REGION Network 4: Block description — Section 3.6 to 4
   // ▂▂▂▂▂▂▂▂▂▂▂▂▂▂▂▂▂▂▂▂▂▂▂▂▂▂▂▂▂▂▂▂▂▂▂▂▂▂▂▂▂▂▂▂
   // 3.6     Operating modes
   // 
   // 
   // This module FC11011_StdDevValve3Way supports various operating modes:
   // 
   //    •   Automatic/manual mode
   // 
   //    •   Interlock bypass mode
   // 
   //    •   Simulation mode
   // 
   //    •   Remote/local mode
   // 
   //    •   Faceplate disabled mode
   // 
   // Examining these in turn:   
   // 
   // 
   // 
   // ▁▁▁▁▁▁▁▁▁▁▁▁▁▁▁▁▁▁▁▁▁▁▁▁▁▁▁▁▁▁▁▁▁▁▁▁▁▁▁▁▁▁▁▁
   // 3.6.1    Automatic and manual modes
   // 
   // 
   // Under normal operation, the valve is in automatic mode and is controlled directly by the 
   // Controller software (usually, sequential or continuous logic); however, it is possible for the 
   // operator to take direct control of the valve by switching it to manual mode.
   // 
   // If manual mode is active, the valve will be energised and deenergised directly at the command 
   // of the operator and will ignore any automatic mode energise and deenergise requests.
   // 
   // If the valve is operating under automatic mode, the manual energise/deenergise request follows 
   // that of the automatic mode; this ensures that the valve remains in the same state when initially 
   // switched from automatic mode to manual mode, referred to as bumpless transfer. This approach 
   // minimises any disturbance to the process should the valve be inadvertently switched to manual 
   // mode.
   // 
   // The following data points are associated with automatic/manual mode:
   // 
   //  DATA STRUCTURE    UT11011_St_DevValve3Way
   //  ――――――――――――――――――――――――――――――――――――――――――
   //  SIGNAL         FUNCTION               TYPE     DETAILS
   //  ――――――――――――――――――――――――――――――――――――――――――
   //  CONFIG_MAN_DIS     Prevents manual mode being       Bool  1 = no manual mode
   //            activated under all circumstances            0 = manual permitted
   //  ――――――――――――――――――――――――――――――――――――――――――
   // 
   //  DATA STRUCTURE    UT31011_Dy_DevValve3Way
   //  ――――――――――――――――――――――――――――――――――――――――――
   //  SIGNAL         FUNCTION               TYPE     DETAILS
   //  ――――――――――――――――――――――――――――――――――――――――――
   //  Mode_AutMan     Identifies the operating mode of     Bool  1 = automatic mode
   //            the valve.                   0 = manual mode
   // 
   //  ctrl_Aut_EngDeng    Causes the valve to energise and         Bool  1 = energise valve
   //            deenergise if auto mode is active          0 = deenergise valve
   // 
   //  ctrl_Man_EngDeng   Causes the valve to energise and         Bool  1 = energise valve
   //            deenergise if man mode is active          0 = deenergise valve
   // 
   //  status_Aut      The valve is in automatic mode      Bool  1 = auto mode
   //                                  0 = no in auto
   // 
   //  status_Man       The valve is in manual mode     Bool  1 = manual mode
   //                                  0 = no in manual
   //  ――――――――――――――――――――――――――――――――――――――――――
   // 
   // Manual mode can only be activated by the operator via a faceplate available at the supervisory 
   // system (SCADA/HMI). 
   // 
   // 
   // 
   // ▁▁▁▁▁▁▁▁▁▁▁▁▁▁▁▁▁▁▁▁▁▁▁▁▁▁▁▁▁▁▁▁▁▁▁▁▁▁▁▁▁▁▁▁
   // 3.6.2    Interlock bypass mode
   // 
   // 
   // All interlock signals (TRIP, INTERLOCK or PERMISSIVE) can be overridden (bypassed). The bypass 
   // signal is a single signal that, if active, overrides and deactivates any TRIP, INTERLOCK or 
   // PERMISSIVE signal that may have been activated.
   // 
   // It is possible to permanently disable the bypass mode for any given valve (preventing the 
   // operator from activating it).
   // 
   // The following data points are associated with the bypass mode:
   // 
   //  DATA STRUCTURE    UT11011_St_DevValve3Way
   //  ――――――――――――――――――――――――――――――――――――――――――
   //  SIGNAL       FUNCTION                TYPE     DETAILS
   //  ――――――――――――――――――――――――――――――――――――――――――
   //  CONFIG_BYPASS_DIS    Prevents bypass mode being      Bool     1 = no bypass mode
   //             activated under all circumstances         0 = bypass permitted
   //  ――――――――――――――――――――――――――――――――――――――――――
   // 
   //  DATA STRUCTURE    UT31011_Dy_DevValve3Way
   //  ――――――――――――――――――――――――――――――――――――――――――
   //  SIGNAL         FUNCTION                TYPE     DETAILS
   //  ――――――――――――――――――――――――――――――――――――――――――
   //  mode_BypassOn   Activates bypass mode, if active, any    Bool     1 = bypass mode on
   //            TRIP, INTERLOCK or PERMISSIVE signal          0 = bypass mode off
   //            will be ignored
   // 
   //  status_BypassOn   Status indication, shows if bypass      Bool     1 = bypass active
   //            mode is active                 0 = bypass inactive
   //  ――――――――――――――――――――――――――――――――――――――――――
   // 
   // Bypass mode can only be activated by the operator usually via a faceplate available at the 
   // supervisory system (SCADA/HMI), alternatively it may be via some form of hardwired signal such 
   // as a key-switch &c. 
   // 
   // If bypass mode is disabled (configuration signal CONFIG_BYPASS_DIS is set to 1), then the bypass 
   // mode cannot be turned on under any circumstances, the option will be greyed out on the 
   // supervisory system faceplate and the module will constantly reset the mode_BypassOn signal.  
   // 
   // 
   // 
   // ▁▁▁▁▁▁▁▁▁▁▁▁▁▁▁▁▁▁▁▁▁▁▁▁▁▁▁▁▁▁▁▁▁▁▁▁▁▁▁▁▁▁▁▁
   // 3.6.3    Simulation mode
   // 
   // 
   // The module can be switched to a simulation mode, in which the position feedback for the valve 
   // is replaced by simulated signals specified by the operator. 
   // 
   // Simulation mode is generally used during testing, but can also be applied in a process 
   // environment if a fault condition is detected; this scenario allows the plant to continue operating 
   // (albeit under some degree of manual control) until the valve is repaired or replaced.
   // 
   // The following data points are associated with the simulation mode:
   // 
   //  DATA STRUCTURE    UT11011_St_DevValve3Way
   //  ――――――――――――――――――――――――――――――――――――――――――
   //  SIGNAL       FUNCTION                TYPE     DETAILS
   //  ――――――――――――――――――――――――――――――――――――――――――
   //  CONFIG_SIM_DIS     Prevents simulation mode being     Bool     1 = no sim mode
   //             activated under all circumstances         0 = sim permitted
   //  ――――――――――――――――――――――――――――――――――――――――――
   //  DATA STRUCTURE    UT31011_Dy_DevValve3Way
   //  ――――――――――――――――――――――――――――――――――――――――――
   //  SIGNAL         FUNCTION                TYPE     DETAILS
   //  ――――――――――――――――――――――――――――――――――――――――――
   //  mode_SimOn      Activates simulation mode, if active, the   Bool     1 = sim mode on
   //            position feedback will be specified by         0 = sim mode off
   //            mode_SimValue      
   //  mode_SimValue    Specifies the type of simulated position     Int     0 = no feedback
   //            feedback in use                  1 = permanently eng
   //                                      2 = permanently deng
   //                                      3 = follow demand
   // 
   //  status_SimOn     Status indication, shows if simulation     Bool     1 = sim active
   //            mode is active                 0 = sim inactive
   //  ――――――――――――――――――――――――――――――――――――――――――
   // 
   // Simulation mode can only be activated by the operator via a faceplate available at the 
   // supervisory system (SCADA/HMI).
   // 
   // If simulation mode is activated, the position feedback for the valve is forced to one of four 
   // states specified by the mode_SimValue variable (this is an enumerated variable):
   // 
   //  ――――――――――――――――――――――――――――――――――――――――――
   //  mode_SimValue  DESCRIPTION                FBK_ENG FBK_DENG
   //  ――――――――――――――――――――――――――――――――――――――――――
   //      0        Permanently disables all position feedback    0     0
   //             (irrespective of any valve position)
   // 
   //      1        Permanently sets valve position to energised         1     0
   //             (irrespective of any valve position)
   // 
   //      2        Permanently sets valve position to deenergised    0     1
   //             (irrespective of any valve position)
   // 
   //      3        Position feedback follows the requested        1/0    0/1
   //             state of the valve                (if valve is eng/deng)
   //  ――――――――――――――――――――――――――――――――――――――――――
   // 
   // The mode_SimValue is restricted to the range 0-3.
   // 
   // If simulation mode is disabled (configuration signal CONFIG_SIM_DIS is set to 1), then the 
   // simulation mode cannot be turned on under any circumstances, the option will be greyed out on 
   // the supervisory system faceplate and the module will constantly reset the mode_SimOn signal.
   // 
   // If simulation mode is permitted (CONFIG_SIM_DIS = 0), then setting mode_SimOn to 1 will activate 
   // simulation mode and the any position feedback signals (connected to FBK_ENG and 
   // FBK_DENG) will be overridden according to the value stored in mode_SimValue (see Table above).
   // 
   // The operator can set and adjust the simulation value (mode_SimValue) from the instrument 
   // faceplate on the supervisory system. The simulation value can be adjusted at any time by the 
   // operator (even if simulation mode has not been activated), but will not be applied until 
   // simulation mode is turned on (mode_SimOn = 1). 
   // 
   // If simulation mode is completely disabled (CONFIG_SIM_DIS is set to 1) then the operator will not 
   // be able to adjust the simulated value (mode_SimValue will be greyed out on the faceplate).
   // 
   // 
   // 
   // ▁▁▁▁▁▁▁▁▁▁▁▁▁▁▁▁▁▁▁▁▁▁▁▁▁▁▁▁▁▁▁▁▁▁▁▁▁▁▁▁▁▁▁▁
   // 3.6.4     Remote/local mode
   // 
   // Remote and local operating modes refer to the supervisory system that has control of the 
   // device (i.e. which system can write to the device and change the operating mode of the 
   // device). 
   // 
   // This type of mode is usual present where a plant has a remote central control location (a control 
   // room) that normally controls the device (remote control), but also has a field panel with a local 
   // HMI that an operator in the field can select to take over control of the device (local control) for 
   // maintenance purposes.
   // 
   // The modes are as follows (and are mutually exclusive, only one will be active):
   // 
   //    Remote        Only the remote system in the control room can 
   //                 control the device
   // 
   //    Local            A local system has taken control of the device and the remote 
   //                 system can no longer issue commands to it
   // 
   //    Remote/local disabled   The system does not use remote/local modes and any 
   //      (ALL mode)     supervisory system can issue commands to the device 
   //  
   // Remote/local control is generally handled by the supervisory systems themselves; however, the 
   // supervisory systems need a storage area per device to record which mode that device is in, local 
   // control is often activated by a panel key-switch, that changes the state of several devices from 
   // remote to local (usually all the devices controlled by the local panel).
   // 
   // The module simply identifies the remote/local mode from the mode signals and configuration 
   // signals provided to the module.
   // 
   // For systems that do not use remote/local modes (any supervisory system can control the device, 
   // or control is determined by operator privileges), the remote/local modes can be disabled 
   // (CONFIG_RL_EN is set to zero) and the device is effectively in ALL mode (any system can 
   // control the device).
   // 
   // If remote/local operation is in use, the supervisory system that does not have control will still 
   // display all the information from the device, but will not be able to control the device (it could not 
   // for example, activate simulation mode) and all control function (faceplate functions) will be 
   // greyed out.
   // 
   // The following signals are associated with remote/local/all modes:
   // 
   //  DATA STRUCTURE    UT11011_St_DevValve3Way
   //  ――――――――――――――――――――――――――――――――――――――――――
   //  SIGNAL           FUNCTION            TYPE   DETAILS
   //  ――――――――――――――――――――――――――――――――――――――――――
   //  CONFIG_RL_EN      Allows Remote and Local      Bool    1 = Remote/local selected
   //                 modes to be selected        0 = All mode is active
   // 
   //  DATA STRUCTURE    UT31011_Dy_DevValve3Way
   //  ――――――――――――――――――――――――――――――――――――――――――
   //  SIGNAL           FUNCTION            TYPE   DETAILS
   //  ――――――――――――――――――――――――――――――――――――――――――
   //  mode_RemoteOn       Activates remote mode     Bool    1 = remote mode on, 
   //                 CONFIG_RL_EN must = 1       0 = remote mode off
   // 
   //  mode_LocalOn     Activates local mode          Bool    1 = local mode on, 
   //                 CONFIG_RL_EN must = 1       0 = remote mode off
   // 
   //  status_RemoteOn      Status remote mode on     Bool    1 = remote mode on, 
   //                               0 = remote mode off
   // 
   //  status_LocalOn       Status local mode on      Bool 1 = local mode on, 
   //                               0 = local mode off
   // 
   //  status_RLOff       Status ALL mode is on = 0    Bool 1 = ALL mode on, 
   //                               0 = ALL mode off
   //  ――――――――――――――――――――――――――――――――――――――――――
   //  Block remote/local signals 
   // 
   // By default, remote/local is disabled — ALL mode is selected (CONFIG_RL_EN = 0).
   // 
   // 
   // 
   // 
   // ▁▁▁▁▁▁▁▁▁▁▁▁▁▁▁▁▁▁▁▁▁▁▁▁▁▁▁▁▁▁▁▁▁▁▁▁▁▁▁▁▁▁▁▁
   // 3.6.5     Faceplate disable mode
   // 
   // It is possible to disable the supervisory system faceplate from within the module, the 
   // configuration signal:
   // 
   // 
   //  ――――――――――――――――――――――――――――――――――――――――――
   //  SIGNAL           FUNCTION            TYPE   DETAILS
   //  ――――――――――――――――――――――――――――――――――――――――――
   //  CONFIG_FP_DIS        Disable the supervisory      Bool    1 = Faceplate disabled
   //                 system faceplate           0 = normal
   //  ――――――――――――――――――――――――――――――――――――――――――
   // 
   // If the faceplate is disabled (CONFIG_FP_DIS = 1), the supervisory system must not allow the 
   // device faceplate to be opened (normally achieved by clicking the block icon or device symbol), 
   // this in turn prevents the operator from affecting the device in anyway, it would not, for example, 
   // be possible to put the device into simulation mode.
   // 
   // Similarly, if the faceplate is disabled, the operator will not have access to the mode_Reset signal, 
   // meaning that alternative reset mechanisms must be in place (such as a hardwired pushbutton 
   // for example).
   // 
   //                ━━━   ⬙⬙⬙⬙⬙⬙   ━━━
   // 
   // 
   // 
   // ▄▄▄▄▄▄▄▄▄▄▄▄▄▄▄▄▄▄▄▄▄▄▄▄▄▄▄▄▄▄▄▄▄▄▄▄▄▄▄▄▄▄▄▄
   // 4.     Supervisory system interface
   // 
   // 
   // See the online documentation for this block — select the block in the project tree and press:
   //      SHIFT + F1 or follow the link: https://psop.uk/pal-smds-fc11011-p 
   // 
   // An explanation of the block icons and faceplates available to the supervisory system for this 
   // module is given in section 4 of the SMDS document [Ref. 011].
   // 
   // A downloadable copy of the SMDS (and all other project documentation) is available here:
   // 
   //      https://practicalseries.com/2001-pal/21-project/01-00-docs.html
   // 
   // For this module, the document number is: PS2001-5-2312-fc11011
   // 
   //                ━━━   ⬙⬙⬙⬙⬙⬙   ━━━
END_REGION

REGION Network 5: Block description — Sections 5 to 11
   // ▄▄▄▄▄▄▄▄▄▄▄▄▄▄▄▄▄▄▄▄▄▄▄▄▄▄▄▄▄▄▄▄▄▄▄▄▄▄▄▄▄▄▄▄
   // 5.     PARAMETERS
   // 
   // 
   // The following parameters are associated with the block:
   // 
   //  
   //  ――――――――――――――――――――――――――――――――――――――――――
   //  PARAM         FUNCTION                    TYPE      IN-OUT 
   //  ――――――――――――――――――――――――――――――――――――――――――
   //  SYS_SIGNALS      Common system signals              UT21000    In
   //           logic and timing signals for parametric access
   // 
   //  FBK_ENG        Optional energised state positive feedback     Bool      In
   //           (1 = energised, 0 = not energised) If not 
   //           required, set permanently to _False
   // 
   //  FBK_DENG     Optional deenergised state positive feedback   Bool      In
   //           (1 = deenergised, 0 = not deenergised) If not  
   //           required, set permanently to _False
   // 
   //  EXT_FAULT     Optional external fault signal for the device     Bool      In
   //           (1 = fault, 0 = healthy). If not required, set 
   //           permanently to _False
   // 
   //  E_STOP        Optional emergency stop (safety) signal        Bool      In
   //           (1 = emergency stop active, 0 = healthy) If not 
   //           required, set permanently to _False
   // 
   //  TRIP        Optional trip signal                  Bool      In
   //           (1 = trip condition active, 0 = healthy) If not 
   //           required, set permanently to _False
   // 
   //  INTERLOCK     Optional interlock signal               Bool      In
   //           (1 = interlock condition active, 0 = healthy) If 
   //           not required, set permanently to _False
   // 
   //  PERMISSIVE      Optional permissive signal             Bool      In
   //           (1 = permissive condition active, 0 = healthy) 
   //           If not required, set permanently to _False
   // 
   //  STATIC_DATA     Data structure that holds the configuration data     UT11011    In
   //           for the device (limit switch and interlock 
   //           configuration &c.)
   // 
   //  DYNAMIC_DATA      Data structure that holds the live data for the       UT31011    InOut
   //           device (its mode, status and messages and 
   //           any other dynamic information required by the 
   //           module)
   // 
   //  OPERATE        Output to drive the valve to a particular state    Bool      Out
   //           (1 = energised state, 0 = deenergised state)
   //  ――――――――――――――――――――――――――――――――――――――――――
   // 
   //                ━━━   ⬙⬙⬙⬙⬙⬙   ━━━
   // 
   // 
   // ▄▄▄▄▄▄▄▄▄▄▄▄▄▄▄▄▄▄▄▄▄▄▄▄▄▄▄▄▄▄▄▄▄▄▄▄▄▄▄▄▄▄▄▄
   // 6.     DATA STRUCTURES AND USAGE
   // 
   // 
   // The block has the following associated data structure:
   // 
   // 
   //  ――――――――――――――――――――――――――――――――――――――――――
   //  DATA STRUCTURE             DESCRIPTION
   //  ――――――――――――――――――――――――――――――――――――――――――
   //  UT01000_St_SysRevision          Revision information for this block    See FC01001
   //  UT01001_St_SysLicence           Licence information for this block  See FC01001
   //  UT21000_Dy_SysSignals           System signals for logic and timing  See FC01001
   // 
   //  UT11011_St_DevValve3Way        Static data that holds the configuration data
   //                     for the device ( limit switch and interlock 
   //                     configuration &c.)
   // 
   //  UT31011_Dy_DevValve3Way          Dynamic data that holds the live data for the
   //                     device (its mode, status and messages and 
   //                     any other dynamic information required by the 
   //                     module)
   // 
   //  ――――――――――――――――――――――――――――――――――――――――――
   // 
   // 
   // 
   // ▂▂▂▂▂▂▂▂▂▂▂▂▂▂▂▂▂▂▂▂▂▂▂▂▂▂▂▂▂▂▂▂▂▂▂▂▂▂▂▂▂▂▂▂
   // 6.1     UT11011_St_DevValve3Way
   // 
   // The static data structure for an isolating valve.
   // 
   // 
   //  UT11011_St_DevValve3Way (full contents)
   //  ――――――――――――――――――――――――――――――――――――――――――
   //  SIGNAL NAME          FUNCTION                     TYPE
   //  ――――――――――――――――――――――――――――――――――――――――――
   //  CONFIG_FBK_ENG_EN      CONFIG — Energised feedback is enabled         Bool
   //                      (1 = energised feedback, 0 = none)
   //  CONFIG_FBK_DENG_EN       CONFIG — Deenergised feedback is enabled       Bool
   //                      (1 = deenergised feedback, 0 = none)
   //  CONFIG_ESTOP_DIS     CONFIG — E_STOP signal disabled           Bool
   //                      (1 = E_STOP not used, 0 = in use)
   //  CONFIG_TRIP_DIS      CONFIG — TRIP signal disabled           Bool
   //                      (1 = TRIP not used, 0 = in use)
   //  CONFIG_ILOCK_DIS     CONFIG — INTERLOCK signal disabled        Bool
   //                      (1 = INTERLOCK not used, 0 = in use)
   //  CONFIG_PERM_DIS      CONFIG — PERMISSIVE signal disabled         Bool
   //                      (1 = PERMISSIVE not used, 0 = in use)
   //  CONFIG_TRIP_ENG_DENG    CONFIG — TRIP state                  Bool
   //                      (1 = energised, 0 = deenergised)
   //  CONFIG_ILOCK_ENG_DENG   CONFIG — INTERLOCK state              Bool
   //                      ((1 = energised, 0 = deenergised)
   //  CONFIG_PERM_ENG_DENG    CONFIG — PERMISSIVE permitted state         Bool
   //                      (1 = energised, 0 = deenergised)
   //  CONFIG_FP_DIS               CONFIG — Faceplate is disabled           Bool
   //                      (1 = no Faceplate, 0 = normal)
   //  CONFIG_MAN_DIS              CONFIG — Manual mode is disabled          Bool
   //                      (1 = no manual mode, 0 = normal)
   //  CONFIG_BYPASS_DIS     CONFIG — Bypass mode is disabled           Bool
   //                      (1 = no bypass mode, 0 = normal)
   //  CONFIG_SIM_DIS             CONFIG — Simulation is disabled            Bool
   //                      (1 = no simulation, 0 = normal)
   //  CONFIG_RL_EN       CONFIG — Remote/local mode enabled       Bool
   //                      (1 = enabled, 0 = all mode)
   // 
   //  INFO_TAG          INFORMATION — Instrument ID tag          String[20]
   // 
   //  TIME_ENG_MAX       TIMER — Initial value of energising operation timer  Real
   //                      (counts down from this value), [seconds]
   //  TIME_DENG_MAX             TIMER — Initial value of deeng'ing operation timer   Real
   //                      (counts down from this value), [seconds]
   //  TIME_DER_ENG                TIMER — Percentage of energising timer to expired     Real
   //                      before simulating FBK_ENG, [percent]
   //  TIME_DER_DENG                TIMER — Percentage of deeng'ing timer to expired   Real
   //                      before simulating FBK_DENG, [percent]
   //  ――――――――――――――――――――――――――――――――――――――――――
   // 
   // 
   // 
   // ▂▂▂▂▂▂▂▂▂▂▂▂▂▂▂▂▂▂▂▂▂▂▂▂▂▂▂▂▂▂▂▂▂▂▂▂▂▂▂▂▂▂▂▂
   // 6.2      UT31011_Dy_DevValve3Way
   // 
   // The static data structure for an isolating valve.
   // 
   // 
   //  UT31011_Dy_DevValve3Way (full contents)
   //  ――――――――――――――――――――――――――――――――――――――――――
   //  SIGNAL NAME          FUNCTION                     TYPE
   //  ――――――――――――――――――――――――――――――――――――――――――
   //  status_Denergised      STATUS — Valve is confirmed deenergised        Bool
   //                      (1 = deenergised, 0 = not deenergised)
   //  status_Energised        STATUS — Valve is confirmed energised         Bool
   //                      (1 = energised, 0 = not energised)
   //  status_Deenergising     STATUS — Valve is deenergising           Bool
   //                      (1 = deenergising, 0 = not deenergising)
   //  status_Energising        STATUS — Valve is energising            Bool
   //                      (1 = energising, 0 = not energising)
   //  status_Operating        STATUS — Valve is changing state           Bool
   //                      (1 = changing state, 0 = fixed state)
   //  status_Fault            STATUS — Valve is in fault              Bool
   //                      (1 = fault present, 0 = healthy)
   //  status_OperateOn      STATUS — Valve output is on              Bool
   //                      (1 = energised, 0 = deenergised)
   //  status_Aut           STATUS — Automatic mode active           Bool
   //                      (1 = auto mode on, 0 = auto mode off)
   //  status_Man          STATUS — Manual mode active             Bool
   //                      (1 = man mode on, 0 = man mode off)
   //  status_EStop          STATUS — E_STOP safety signal is active         Bool
   //                      (1 = active, 0 = healthy)
   //  status_Trip        STATUS — TRIP signal is active             Bool
   //                      (1 = active, 0 = healthy)
   //  status_Ilock         STATUS — INTERLOCK signal is active            Bool
   //                      (1 = active, 0 = healthy)
   //  status_Perm        STATUS — PERMISSIVE signal is active           Bool
   //                      (1 = active, 0 = healthy)
   //  status_BypassOn        STATUS — Valve is in bypass mode          Bool
   //                      (1 = Simulation mode, 0 = normal)
   //  status_SimOn           STATUS — Valve is in simulation mode               Bool
   //                      (1 = Simulation mode, 0 = normal)
   //  status_RemoteOn       STATUS — Valve is in remote mode                  Bool
   //                      (1 = Remote mode, 0 = normal)
   //  status_LocalOn         STATUS — Valve is in local mode                    Bool
   //                      (1 = Local mode, 0 = normal)
   //  status_RLOff         STATUS — Valve is in ALL mode                   Bool
   //                      (1 = ALL mode, 0 = normal)
   // 
   //  msg_FailToEnergise       MESSAGE — Alarm – “Fail to energise” active      Bool
   //  msg_FailToDeenergise     MESSAGE — Alarm – “Fail to deenergise” active    Bool
   //  msg_FailWhileEnergised     MESSAGE — Alarm – “Fail while energised” active    Bool
   //  msg_FailWhileDeenergised   MESSAGE — Alarm – “Fail while deenergised” active  Bool
   //  msg_Flt_External         MESSAGE — Alarm – “external fault" is active      Bool
   // 
   //  mode_AutMan        MODE — Automatic or manual mode selection     Bool
   //                    (1 = auto mode active, 0 = man mode)
   //  mode_BypassOn      MODE — Bypass mode                Bool
   //                    (1 = bypass mode active, 0 = normal)
   //  mode_SimOn         MODE — Simulation mode               Bool
   //                    (1 = sim mode active, 0 = normal)
   //  mode_SimValue       MODE — Simulation value               Int
   //                    (0 = no limits, 1 = always eng, 
   //                    2 = always deng, 3 = follow demand)
   //  mode_RemoteOn        MODE — Remote SCADA control enabled       Bool
   //                    (1 = active, 0 = disabled or N/A)
   //  mode_LocalOn         MODE — Local HMI control enabled           Bool
   //                    (1 = active, 0 = disabled or N/A)
   //  mode_Reset        MODE — Fault reset – 1 cycle only           Bool
   //                    (1 = Reset faults, 0 = does nothing)
   //  ctrl_Aut_EngDeng       CONTROL — Auto mode operate the valve      Bool
   //                          (1 = energise, 0 = deenergise)
   //  ctrl_Man_EngDeng         CONTROL — Manual mode operate the valve       Bool
   //                          (1 = energise, 0 = deenergise)
   // 
   //  batch_ID         BATCH — Booking ID (optional for batch operations)   UInt
   // 
   //  actual_Operating_Timer     ACTUAL — Timer value — operating timer      Real
   //                      actual value [seconds]
   //  actual_Last_Op_Time       ACTUAL — actual time taken to achieve the last    Real
   //                      good valve position [seconds]
   // 
   //  $derived_fbk_eng       INTERNAL — Derived feedback energise signal       Bool
   //                          (1 = eng , 0 = not eng)
   //  $derived_fbk_deng         INTERNAL — Derived feedback deenergised signal   Bool
   //                          (1 = deng, 0 = not deng)
   //  $sim_fbk_eng           INTERNAL — Simulated feedback energised signal      Bool
   //                          (1 = eng , 0 = not eng)
   //  $sim_fbk_deng             INTERNAL — Simulated feedback deenergised signal Bool
   //                          (1 = deng, 0 = not deng)
   //  $ctrl_EngDeng           INTERNAL — actual eng or deng request,            Bool
   //                          incorporates all priorities
   //                         (1 = eng valve, 0 = deng valve)
   //  $pret_eng                INTERNAL — Edge retention (+ve) rising edge of    Bool
   //                          ctrl_EngDeng (change to eng)
   //  $nret_deng             INTERNAL — Edge retention (-ve) falling edge of        Bool
   //                          ctrl_EngDeng (change to deng)
   //  ――――――――――――――――――――――――――――――――――――――――――
   // 
   // 
   // With the exception of the flowing, all these signals are discussed in the previous sections, the 
   // outstanding items are firstly:
   // 
   //      batch_ID
   // 
   // The batch_ID is not required for normal use; it is only used where a “booking” system is used 
   // (common in batch and routing applications). Such booking applications can acquire the device 
   // if it is free and reserve it for a particular phase of the batch. Batch applications are a topic in 
   // their own right and are discussed separately in the online User Guide.
   // 
   // There are internal working signals (all signals the start with a $ are internal working signals used 
   // by the module). In this instance they are used as follows: 
   //  
   // The $derived_fbk_eng and $derived_fbk_deng are the internally derived energised and 
   // deenergised feedback signal used in place of FBK_ENG and FBK_DENG if either 
   // CONFIG_FBK_ENG_EN or CONFIG_FBK_DENG_EN is set to zero.
   // 
   // The $sim_fbk_eng and $sim_fbk_deng are the simulated position feedback signal used in place 
   // of FBK_ENG and FBK_DENG if simulation mode is active.
   // 
   // $ctrl_EngDeng is the required state of the valve, it takes into account the auto/manual requested 
   // state and modifies this according to any interlocks, safety signals or faults that may be present.
   // 
   // The $pret_eng and $nret_deng are edge retention signals used to detect either a rising 
   // (a change to energising) or a falling (a change to deenergising) edge on the 
   // $ctrl_EngDeng signal.
   // 
   // 
   //                ━━━   ⬙⬙⬙⬙⬙⬙   ━━━
   // 
   // 
   // 
   // ▄▄▄▄▄▄▄▄▄▄▄▄▄▄▄▄▄▄▄▄▄▄▄▄▄▄▄▄▄▄▄▄▄▄▄▄▄▄▄▄▄▄▄▄
   // 7.     CONSTANTS AND TEMPORARY (LOCAL) DATA
   // 
   // 
   // 
   // ▂▂▂▂▂▂▂▂▂▂▂▂▂▂▂▂▂▂▂▂▂▂▂▂▂▂▂▂▂▂▂▂▂▂▂▂▂▂▂▂▂▂▂▂
   // 7.1     Constants
   // 
   // 
   // The following constants data is used:
   // 
   //  ――――――――――――――――――――――――――――――――――――――――――
   //  SIGNAL NAME       Value    FUNCTION                  TYPE
   //  ――――――――――――――――――――――――――――――――――――――――――
   //  k_TIME_OP_MIN      0.21      Minimum value for the operation timer     Real
   //  ――――――――――――――――――――――――――――――――――――――――――
   // 
   // 
   // 
   // ▂▂▂▂▂▂▂▂▂▂▂▂▂▂▂▂▂▂▂▂▂▂▂▂▂▂▂▂▂▂▂▂▂▂▂▂▂▂▂▂▂▂▂▂
   // 7.2     Temporary (local) data
   // 
   // 
   // The following temporary data is used:
   // 
   //  ――――――――――――――――――――――――――――――――――――――――――
   //  SIGNAL NAME          FUNCTION                  TYPE
   //  ――――――――――――――――――――――――――――――――――――――――――
   //  revInfo             Revision information for the block         UT01000
   //  licInfo           Licensing information for the block      UT01001
   //  calDengElapsedTime          Calc - Derived deng signal elapsed time      Real
   //  calEngElapsedTime       Calc - Derived eng signal elapsed time     Real
   //  wrkEng               Working - eng position feedback signal        Bool
   //  wrkDeng           Working - deng position feedback signal      Bool
   //  wrkCtrlPriority40        Working - priority 40 controls the valve      Bool
   //  wrkCtrlPriority30        Working - priority 30 controls the valve      Bool
   //  wrkCtrlPriority20        Working - priority 20 controls the valve      Bool
   //  wrkCtrlPriority10        Working - priority 10 controls the valve      Bool
   //  wrkCtrlPriority00        Working - priority 00 controls the valve      Bool
   //  wrkCtrlAutManEngDeng   Working - aut/man eng or deng request        Bool
   //  wrkTimeFbkEngSim        Working - Err checked TIME_DER_ENG                 Real
   //  wrkTimeFbkDengSim       Working - Err checked TIME_DER_DENG              Real
   //  wrkInt           Working storage area (integer)          Int
   //  wrkReal           Working storage (Real)             Real
   //  wrkDInt           Working storage area (double integer)         DInt
   //  ――――――――――――――――――――――――――――――――――――――――――
   // 
   //                ━━━   ⬙⬙⬙⬙⬙⬙   ━━━
   // 
   // 
   // 
   // ▄▄▄▄▄▄▄▄▄▄▄▄▄▄▄▄▄▄▄▄▄▄▄▄▄▄▄▄▄▄▄▄▄▄▄▄▄▄▄▄▄▄▄▄
   // 8.     BLOCK CALLS AND ASSOCIATIONS
   // 
   // 
   // This section details any blocks which may be called from within this software module (subroutine 
   // functions for example), any partner blocks with which it may be associated (for example a 
   // receive module that is partner with a transmit module &c.). It lists any system functions which 
   // may be called (e.g. reading the real time clock) and any system data types that may be used.
   // 
   // Finally, it lists any special calling requirements for the block (for example, must be called from 
   // within a cyclic interrupt organisation block) and if the block is using “optimised access” (this is 
   // the default arrangement).
   // 
   // 
   // 
   // ▂▂▂▂▂▂▂▂▂▂▂▂▂▂▂▂▂▂▂▂▂▂▂▂▂▂▂▂▂▂▂▂▂▂▂▂▂▂▂▂▂▂▂▂
   // 8.1     Block calls from within this module
   // 
   // 
   // There are no PAL block calls from within this block.
   // 
   // 
   // 
   // ▂▂▂▂▂▂▂▂▂▂▂▂▂▂▂▂▂▂▂▂▂▂▂▂▂▂▂▂▂▂▂▂▂▂▂▂▂▂▂▂▂▂▂▂
   // 8.2     Blocks associated with this module
   // 
   // 
   // This is a stand-alone block and is not associated with any other blocks.
   // 
   // 
   // 
   // ▂▂▂▂▂▂▂▂▂▂▂▂▂▂▂▂▂▂▂▂▂▂▂▂▂▂▂▂▂▂▂▂▂▂▂▂▂▂▂▂▂▂▂▂
   // 8.3     System block calls and system data types
   // 
   // There are no system block calls
   // 
   // 
   // 
   // ▂▂▂▂▂▂▂▂▂▂▂▂▂▂▂▂▂▂▂▂▂▂▂▂▂▂▂▂▂▂▂▂▂▂▂▂▂▂▂▂▂▂▂▂
   // 8.4     Special properties and requirements
   // 
   // 
   // 
   // ▁▁▁▁▁▁▁▁▁▁▁▁▁▁▁▁▁▁▁▁▁▁▁▁▁▁▁▁▁▁▁▁▁▁▁▁▁▁▁▁▁▁▁▁
   // 8.4.1     Block optimisation, IEC compatibility and library conformance
   // 
   // 
   //    •   Block optimisation is ACTIVE for this block.
   // 
   //    •   The block has been checked for IEC compatibility and is compliant.
   // 
   //    •   The block is compatible with all IEC library-conformance module constraints
   // 
   // 
   // 
   // ▁▁▁▁▁▁▁▁▁▁▁▁▁▁▁▁▁▁▁▁▁▁▁▁▁▁▁▁▁▁▁▁▁▁▁▁▁▁▁▁▁▁▁▁
   // 8.4.2     Calling requirements
   // 
   // 
   // There are no special calling requirements for this block.
   // 
   //                ━━━   ⬙⬙⬙⬙⬙⬙   ━━━
   // 
   // 
   // 
   // ▄▄▄▄▄▄▄▄▄▄▄▄▄▄▄▄▄▄▄▄▄▄▄▄▄▄▄▄▄▄▄▄▄▄▄▄▄▄▄▄▄▄▄▄
   // 9.     EXAMPLE USAGE
   // 
   // 
   // The following shows a typical deployment of FC11011:
   // 
   //                         ┌─────────────
   //      ───────────────────┤ FC11011 
   //                         ├───────────────┤
   //    "DB21001_DY_StdGlobalData".SysSignals ─┤ SYS_SIGNALS            %Q1.0
   //                         │             OPERATE ├─  "V001_OPR"
   //                   %I1.2     │               │
   //                "V001_FBK_PORT2" ─┤ FBK_ENG               │
   //                         │               │
   //                   %I1.1     │               │
   //                   "V001_FBK_PORT1" ─┤ FBK_DENG                │
   //                         │               │
   //            %I1.0            │               │
   //           "V001_FAULT"             │               │
   //        ────┤╱├──────────┤ EXT_FAULT                │
   //                         │               │
   //            %I1.4            │               │
   //          "ZONEA_ESTOP"               │               │
   //        ────┤╱├──────────┤ E_STOP                │
   //                         │               │
   //                    "_False" ─┤ TRIP                    │
   //                         │               │
   //            "DB23002_Dy_ILock.V001"─┤ INTERLOCK             │
   //                         │               │
   //                    "_False" ─┤ PERMISSIVE            │
   //                         │               │
   //                         │               │
   //                         │               │
   //         "DB11011_St_DevValve3Way".V001 ─┤ STATIC_DATA             │
   //                         │
   //         "DB31011_Dy_DevValve3Way".V001 ─┤ DYNAMIC_DATA
   //                         │
   //                         │
   //                                         │
   //                                ─────────┘
   // 
   // 
   //               ━━━   ⬙⬙⬙⬙⬙⬙   ━━━
   // 
   // 
   // 
   // ▄▄▄▄▄▄▄▄▄▄▄▄▄▄▄▄▄▄▄▄▄▄▄▄▄▄▄▄▄▄▄▄▄▄▄▄▄▄▄▄▄▄▄▄
   // 10.     TEST AND VERIFICATION PATH
   // 
   // 
   // The following diagram shows the full test and verification path for the formal release of each 
   // version of the software module. See the Test Plan [Ref. 003] for full details, available here:
   //         https://psop.uk/pal-tp-p
   // 
   // 
   //         FC11011-T001         
   // 
   //     Test version: 000.801     
   //  Released version: 001.000     
   // Released commit: D0015    
   // 
   //        SCR      SMT     
   // ＿＿＿＿＿＿┌┐＿＿ ▛▜ ＿＿
   //       └┘   ▙▟   
   // Initial test           
   // 
   // Initial test to release the      
   // module following the      
   // development stage.       
   // Full SMT    
   //           
   // 
   // Where:
   // ――――――――――――――――――――――――――――――――――――――――――――
   //  SCR    Source Code Review      A visual inspection of the software to ensure it has been written  
   // ┌┐             to the correct standards, uses the correct structures within the
   // └┘             software and is generally suitable for deployment.               
   // 
   //  SMT Software Module Test    A full and detailed test of an individual software module in
   //   ▛▜              isolation; such testing requires that all branches of the 
   //   ▙▟              software are tested. 
   // 
   //                It tests all the interfaces to the module, any data recorded or 
   //                stored by the module, all error and exception handling functions 
   //                and tests all timed and interrupt driven operations.
   // 
   //  SCV Software Compatibility     A mechanism for verifying that no executable code software 
   // ╓╖    Verification          changes have been made to a module following changes to
   // ╙╜             comment fields.
   // 
   //                Allows typographical errors &c. to be corrected without forcing 
   //                a full SMT on a module that has not functionally changed.
   // ――――――――――――――――――――――――――――――――――――――――――――
   // 
   // An SCV can only be performed on a module that has at some point previously, successfully 
   // completed both an SCR and SMT. Where an SCV is implemented, it replaces the requirement for 
   // both the SCR and the SMT for the test iteration in question.
   // 
   //                ━━━   ⬙⬙⬙⬙⬙⬙   ━━━
   // 
   // 
   // ██████████████ █ █ █ █  END   █ █ █ █ ██████████████
END_REGION

REGION Network 6: Current revision and modification history
   // ▄▄▄▄▄▄▄▄▄▄▄▄▄▄▄▄▄▄▄▄▄▄▄▄▄▄▄▄▄▄▄▄▄▄▄▄▄▄▄▄▄▄▄▄
   // MODIFICATION HISTORY
   // 
   // 
   // The revision data shown here, in the network comments, contains additional information 
   // reflecting the software development workflow under the version control system (VCS) employed 
   // to track all software changes.
   // 
   // The VCS in use is the Git Source Code Management system in conjunction with the GitHub online 
   // hosting system. The software in its entirety is available in the GitHub remote repository:
   // 
   //      https://github.com/practicalseries/PS2001-pal-software
   // 
   // The repository is public and can be freely copied (forked in GitHub terminology) and used 
   // under the MIT licence. 
   // 
   // The MIT licence is reproduced in full in the last network of this software module.
   // 
   // 
   //  ―――――――――――――――――――――――――――――――――――――――――――
   //  DATE       REVISION             MASTER BRANCH     DEV
   //          (nnn.amm)   COMMIT TAG    (Base ---> Merge)    BRANCH   Author
   //  ———————————————————————————————————————————
   //  2022.06.07    000.801   D0014A-000.801   D0014 N/A     D0014A   M. Gledhill
   //                        Released for test (SMTS)
   // 
   //  2022.06.01    000.101   D0014A-000.101   D0014 N/A     D0014A   M. Gledhill
   //                        Block created
   //  ———————————————————————————————————————————
   //   Where: nnn  =  Major revision
   //         a  =  Type (1-7 Development, 8 Proving, 9 Qualification, 0 Release)
   //       mm  =  Minor revision (must be 00 if a = 0)
   //         Block properties version number should be set to nn.a (only one decimal place)
   // 
   // ▄▄▄▄▄▄▄▄▄▄▄▄▄▄▄▄▄▄▄▄▄▄▄▄▄▄▄▄▄▄▄▄▄▄▄▄▄▄▄▄▄▄▄▄
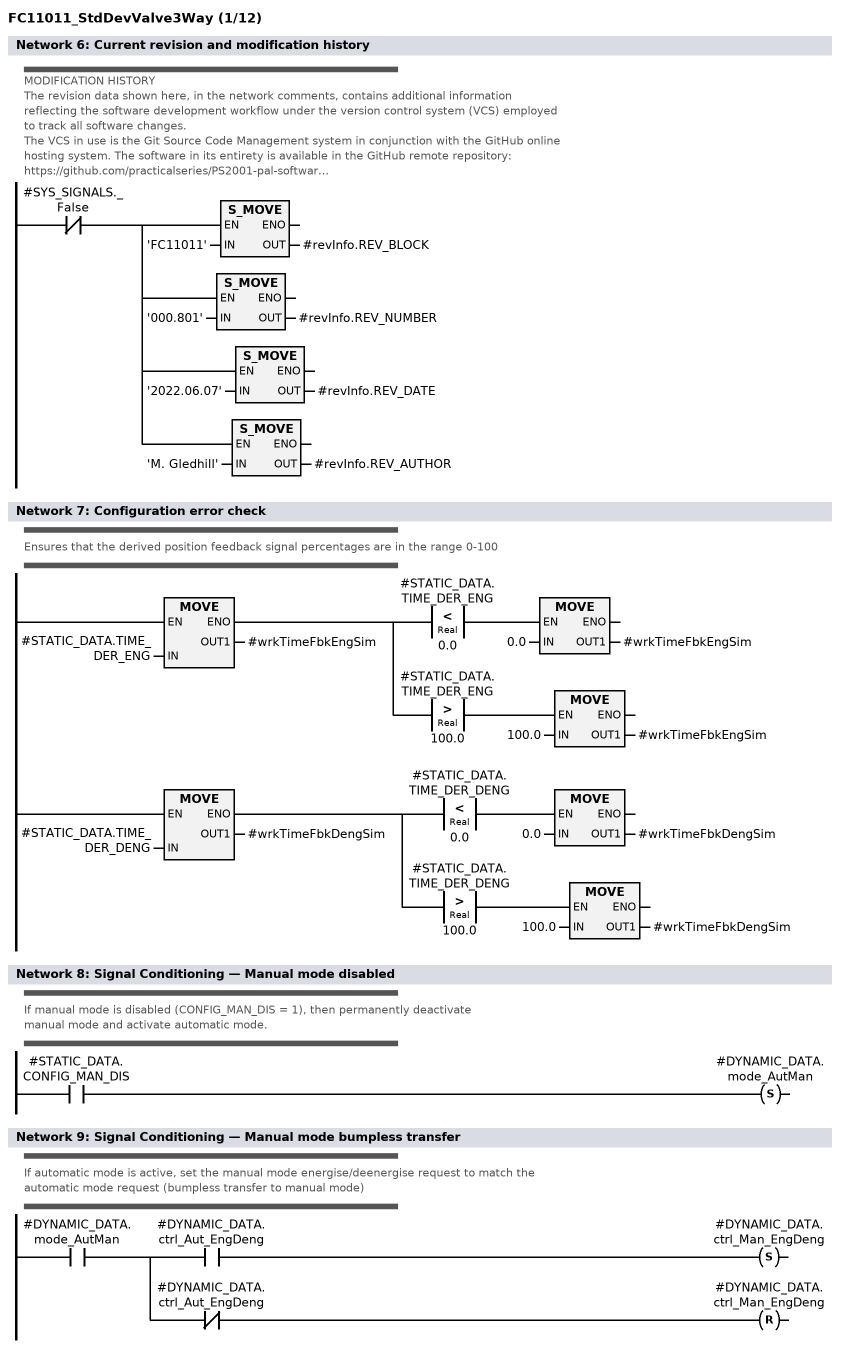
   RUNG wire#powerrail
      I_Contact( #SYS_SIGNALS._False )
      wire#w1
      S_Move(in := 'FC11011', out => #revInfo.REV_BLOCK)
   END_RUNG
   RUNG wire#w1
      S_Move(in := '000.801', out => #revInfo.REV_NUMBER)
   END_RUNG
   RUNG wire#w1
      S_Move(in := '2022.06.07', out => #revInfo.REV_DATE)
   END_RUNG
   RUNG wire#w1
      S_Move(in := 'M. Gledhill', out => #revInfo.REV_AUTHOR)
   END_RUNG
   // the same network as SCL:
   IF NOT #SYS_SIGNALS._False THEN
       #revInfo.REV_BLOCK := 'FC11011';
       #revInfo.REV_NUMBER := '000.801';
       #revInfo.REV_DATE := '2022.06.07';
       #revInfo.REV_AUTHOR := 'M. Gledhill';
   END_IF;
END_REGION

REGION Network 7: Configuration error check
   // ▀▀▀▀▀▀▀▀▀▀▀▀▀▀▀▀▀▀▀▀▀▀▀▀▀▀▀▀▀▀▀▀▀▀▀▀▀▀▀▀▀▀▀▀
   // Ensures that the derived position feedback signal percentages are in the range 0-100
   // ▄▄▄▄▄▄▄▄▄▄▄▄▄▄▄▄▄▄▄▄▄▄▄▄▄▄▄▄▄▄▄▄▄▄▄▄▄▄▄▄▄▄▄▄
   RUNG wire#powerrail
      Move(in := #STATIC_DATA.TIME_DER_ENG, out1 => #wrkTimeFbkEngSim)
      wire#w1
      { S7_Templates := "SrcType := Real" } LT_Contact(in1 := #STATIC_DATA.TIME_DER_ENG, in2 := 0.0)
      Move(in := 0.0, out1 => #wrkTimeFbkEngSim)
   END_RUNG
   RUNG wire#w1
      { S7_Templates := "SrcType := Real" } GT_Contact(in1 := #STATIC_DATA.TIME_DER_ENG, in2 := 100.0)
      Move(in := 100.0, out1 => #wrkTimeFbkEngSim)
   END_RUNG
   RUNG wire#powerrail
      Move(in := #STATIC_DATA.TIME_DER_DENG, out1 => #wrkTimeFbkDengSim)
      wire#w2
      { S7_Templates := "SrcType := Real" } LT_Contact(in1 := #STATIC_DATA.TIME_DER_DENG, in2 := 0.0)
      Move(in := 0.0, out1 => #wrkTimeFbkDengSim)
   END_RUNG
   RUNG wire#w2
      { S7_Templates := "SrcType := Real" } GT_Contact(in1 := #STATIC_DATA.TIME_DER_DENG, in2 := 100.0)
      Move(in := 100.0, out1 => #wrkTimeFbkDengSim)
   END_RUNG
   // the same network as SCL:
   #wrkTimeFbkEngSim := #STATIC_DATA.TIME_DER_ENG;
   IF #STATIC_DATA.TIME_DER_ENG < 0.0 THEN #wrkTimeFbkEngSim := 0.0; END_IF;
   IF #STATIC_DATA.TIME_DER_ENG > 100.0 THEN #wrkTimeFbkEngSim := 100.0; END_IF;
   #wrkTimeFbkDengSim := #STATIC_DATA.TIME_DER_DENG;
   IF #STATIC_DATA.TIME_DER_DENG < 0.0 THEN #wrkTimeFbkDengSim := 0.0; END_IF;
   IF #STATIC_DATA.TIME_DER_DENG > 100.0 THEN #wrkTimeFbkDengSim := 100.0; END_IF;
END_REGION

REGION Network 8: Signal Conditioning — Manual mode disabled
   // ▀▀▀▀▀▀▀▀▀▀▀▀▀▀▀▀▀▀▀▀▀▀▀▀▀▀▀▀▀▀▀▀▀▀▀▀▀▀▀▀▀▀▀▀
   // If manual mode is disabled (CONFIG_MAN_DIS = 1), then permanently deactivate
   // manual mode and activate automatic mode.
   // ▄▄▄▄▄▄▄▄▄▄▄▄▄▄▄▄▄▄▄▄▄▄▄▄▄▄▄▄▄▄▄▄▄▄▄▄▄▄▄▄▄▄▄▄
   RUNG wire#powerrail
      Contact( #STATIC_DATA.CONFIG_MAN_DIS )
      S_Coil( #DYNAMIC_DATA.mode_AutMan )
   END_RUNG
   // the same network as SCL:
   IF #STATIC_DATA.CONFIG_MAN_DIS THEN #DYNAMIC_DATA.mode_AutMan := TRUE; END_IF;
END_REGION

REGION Network 9: Signal Conditioning — Manual mode bumpless transfer
   // ▀▀▀▀▀▀▀▀▀▀▀▀▀▀▀▀▀▀▀▀▀▀▀▀▀▀▀▀▀▀▀▀▀▀▀▀▀▀▀▀▀▀▀▀
   // If automatic mode is active, set the manual mode energise/deenergise request to match the 
   // automatic mode request (bumpless transfer to manual mode)
   // ▄▄▄▄▄▄▄▄▄▄▄▄▄▄▄▄▄▄▄▄▄▄▄▄▄▄▄▄▄▄▄▄▄▄▄▄▄▄▄▄▄▄▄▄
   RUNG wire#powerrail
      Contact( #DYNAMIC_DATA.mode_AutMan )
      wire#w1
      Contact( #DYNAMIC_DATA.ctrl_Aut_EngDeng )
      S_Coil( #DYNAMIC_DATA.ctrl_Man_EngDeng )
   END_RUNG
   RUNG wire#w1
      I_Contact( #DYNAMIC_DATA.ctrl_Aut_EngDeng )
      R_Coil( #DYNAMIC_DATA.ctrl_Man_EngDeng )
   END_RUNG
   // the same network as SCL:
   IF #DYNAMIC_DATA.mode_AutMan AND #DYNAMIC_DATA.ctrl_Aut_EngDeng THEN
       #DYNAMIC_DATA.ctrl_Man_EngDeng := TRUE;
   END_IF;
   IF #DYNAMIC_DATA.mode_AutMan AND NOT #DYNAMIC_DATA.ctrl_Aut_EngDeng THEN
       #DYNAMIC_DATA.ctrl_Man_EngDeng := FALSE;
   END_IF;
END_REGION

REGION Network 10: Signal Conditioning — Bypass mode disabled
   // ▀▀▀▀▀▀▀▀▀▀▀▀▀▀▀▀▀▀▀▀▀▀▀▀▀▀▀▀▀▀▀▀▀▀▀▀▀▀▀▀▀▀▀▀
   // If bypass mode is disabled (CONFIG_BYPASS_DIS = 1), then permanently deactivate
   // bypass mode.
   // ▄▄▄▄▄▄▄▄▄▄▄▄▄▄▄▄▄▄▄▄▄▄▄▄▄▄▄▄▄▄▄▄▄▄▄▄▄▄▄▄▄▄▄▄
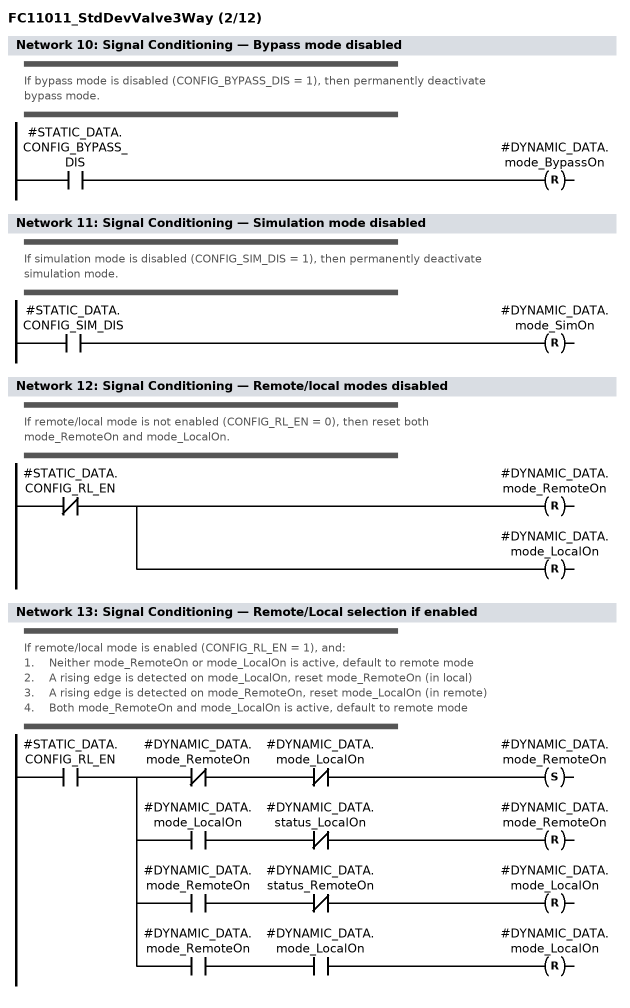
   RUNG wire#powerrail
      Contact( #STATIC_DATA.CONFIG_BYPASS_DIS )
      R_Coil( #DYNAMIC_DATA.mode_BypassOn )
   END_RUNG
   // the same network as SCL:
   IF #STATIC_DATA.CONFIG_BYPASS_DIS THEN #DYNAMIC_DATA.mode_BypassOn := FALSE; END_IF;
END_REGION

REGION Network 11: Signal Conditioning — Simulation mode disabled
   // ▀▀▀▀▀▀▀▀▀▀▀▀▀▀▀▀▀▀▀▀▀▀▀▀▀▀▀▀▀▀▀▀▀▀▀▀▀▀▀▀▀▀▀▀
   // If simulation mode is disabled (CONFIG_SIM_DIS = 1), then permanently deactivate
   // simulation mode.
   // ▄▄▄▄▄▄▄▄▄▄▄▄▄▄▄▄▄▄▄▄▄▄▄▄▄▄▄▄▄▄▄▄▄▄▄▄▄▄▄▄▄▄▄▄
   RUNG wire#powerrail
      Contact( #STATIC_DATA.CONFIG_SIM_DIS )
      R_Coil( #DYNAMIC_DATA.mode_SimOn )
   END_RUNG
   // the same network as SCL:
   IF #STATIC_DATA.CONFIG_SIM_DIS THEN #DYNAMIC_DATA.mode_SimOn := FALSE; END_IF;
END_REGION

REGION Network 12: Signal Conditioning — Remote/local modes disabled
   // ▀▀▀▀▀▀▀▀▀▀▀▀▀▀▀▀▀▀▀▀▀▀▀▀▀▀▀▀▀▀▀▀▀▀▀▀▀▀▀▀▀▀▀▀
   // If remote/local mode is not enabled (CONFIG_RL_EN = 0), then reset both 
   // mode_RemoteOn and mode_LocalOn.
   // ▄▄▄▄▄▄▄▄▄▄▄▄▄▄▄▄▄▄▄▄▄▄▄▄▄▄▄▄▄▄▄▄▄▄▄▄▄▄▄▄▄▄▄▄
   RUNG wire#powerrail
      I_Contact( #STATIC_DATA.CONFIG_RL_EN )
      wire#w1
      R_Coil( #DYNAMIC_DATA.mode_RemoteOn )
   END_RUNG
   RUNG wire#w1
      R_Coil( #DYNAMIC_DATA.mode_LocalOn )
   END_RUNG
   // the same network as SCL:
   IF NOT #STATIC_DATA.CONFIG_RL_EN THEN
       #DYNAMIC_DATA.mode_RemoteOn := FALSE;
       #DYNAMIC_DATA.mode_LocalOn := FALSE;
   END_IF;
END_REGION

REGION Network 13: Signal Conditioning — Remote/Local selection if enabled
   // ▀▀▀▀▀▀▀▀▀▀▀▀▀▀▀▀▀▀▀▀▀▀▀▀▀▀▀▀▀▀▀▀▀▀▀▀▀▀▀▀▀▀▀▀
   // If remote/local mode is enabled (CONFIG_RL_EN = 1), and:
   // 
   //    1.  Neither mode_RemoteOn or mode_LocalOn is active, default to remote mode
   //    2.  A rising edge is detected on mode_LocalOn, reset mode_RemoteOn (in local)
   //    3.  A rising edge is detected on mode_RemoteOn, reset mode_LocalOn (in remote)
   //    4.  Both mode_RemoteOn and mode_LocalOn is active, default to remote mode
   // ▄▄▄▄▄▄▄▄▄▄▄▄▄▄▄▄▄▄▄▄▄▄▄▄▄▄▄▄▄▄▄▄▄▄▄▄▄▄▄▄▄▄▄▄
   RUNG wire#powerrail
      Contact( #STATIC_DATA.CONFIG_RL_EN )
      wire#w1
      I_Contact( #DYNAMIC_DATA.mode_RemoteOn )
      I_Contact( #DYNAMIC_DATA.mode_LocalOn )
      S_Coil( #DYNAMIC_DATA.mode_RemoteOn )
   END_RUNG
   RUNG wire#w1
      Contact( #DYNAMIC_DATA.mode_LocalOn )
      I_Contact( #DYNAMIC_DATA.status_LocalOn )
      R_Coil( #DYNAMIC_DATA.mode_RemoteOn )
   END_RUNG
   RUNG wire#w1
      Contact( #DYNAMIC_DATA.mode_RemoteOn )
      I_Contact( #DYNAMIC_DATA.status_RemoteOn )
      R_Coil( #DYNAMIC_DATA.mode_LocalOn )
   END_RUNG
   RUNG wire#w1
      Contact( #DYNAMIC_DATA.mode_RemoteOn )
      Contact( #DYNAMIC_DATA.mode_LocalOn )
      R_Coil( #DYNAMIC_DATA.mode_LocalOn )
   END_RUNG
   // the same network as SCL:
   IF #STATIC_DATA.CONFIG_RL_EN AND NOT #DYNAMIC_DATA.mode_RemoteOn AND NOT #DYNAMIC_DATA.mode_LocalOn THEN
       #DYNAMIC_DATA.mode_RemoteOn := TRUE;
   END_IF;
   IF #STATIC_DATA.CONFIG_RL_EN AND #DYNAMIC_DATA.mode_LocalOn AND NOT #DYNAMIC_DATA.status_LocalOn THEN
       #DYNAMIC_DATA.mode_RemoteOn := FALSE;
   END_IF;
   IF #STATIC_DATA.CONFIG_RL_EN AND #DYNAMIC_DATA.mode_RemoteOn AND NOT #DYNAMIC_DATA.status_RemoteOn THEN
       #DYNAMIC_DATA.mode_LocalOn := FALSE;
   END_IF;
   IF #STATIC_DATA.CONFIG_RL_EN AND #DYNAMIC_DATA.mode_RemoteOn AND #DYNAMIC_DATA.mode_LocalOn THEN
       #DYNAMIC_DATA.mode_LocalOn := FALSE;
   END_IF;
END_REGION

REGION Network 14: Signal Conditioning — Derived energised position
   // ▀▀▀▀▀▀▀▀▀▀▀▀▀▀▀▀▀▀▀▀▀▀▀▀▀▀▀▀▀▀▀▀▀▀▀▀▀▀▀▀▀▀▀▀
   // If there is no energised position feedback (CONFIG_FBK_ENG_EN = 0), then the energised state 
   // of the valve is derived from the elapsed time of the operation timer using the following 
   // formulae:
   // 
   // ┌───────────────────────────────────────┐
   // │$derived_fbk_eng = 1 when:                             │
   // │                              wrkTimeFbkEngSim    │
   // │actual_Operating_Timer ≤ TIME_ENG_MAX ─ TIME_ENG_MAX ╳ ---------------------------------------- │
   // │                                 100        │
   // └───────────────────────────────────────┘
   // Note:    wrkTimeFbkEngSim is the error checked equivalent of TIME_DER_ENG
   // 
   // If the calculated elapsed time is close to or less than k_TIME_OP_MIN (210ms),
   // the calculated elapsed time (calEngElapsedTime) is set to k_TIME_OP_MIN. This ensures at
   // least one timing pulse is required before the timer reaches zero.
   // 
   // The derived energised signal ($derived_fbk_eng) is reset if the valve is requested to be 
   // deenergised ($ctrl_EngDeng = 0).
   // ▄▄▄▄▄▄▄▄▄▄▄▄▄▄▄▄▄▄▄▄▄▄▄▄▄▄▄▄▄▄▄▄▄▄▄▄▄▄▄▄▄▄▄▄
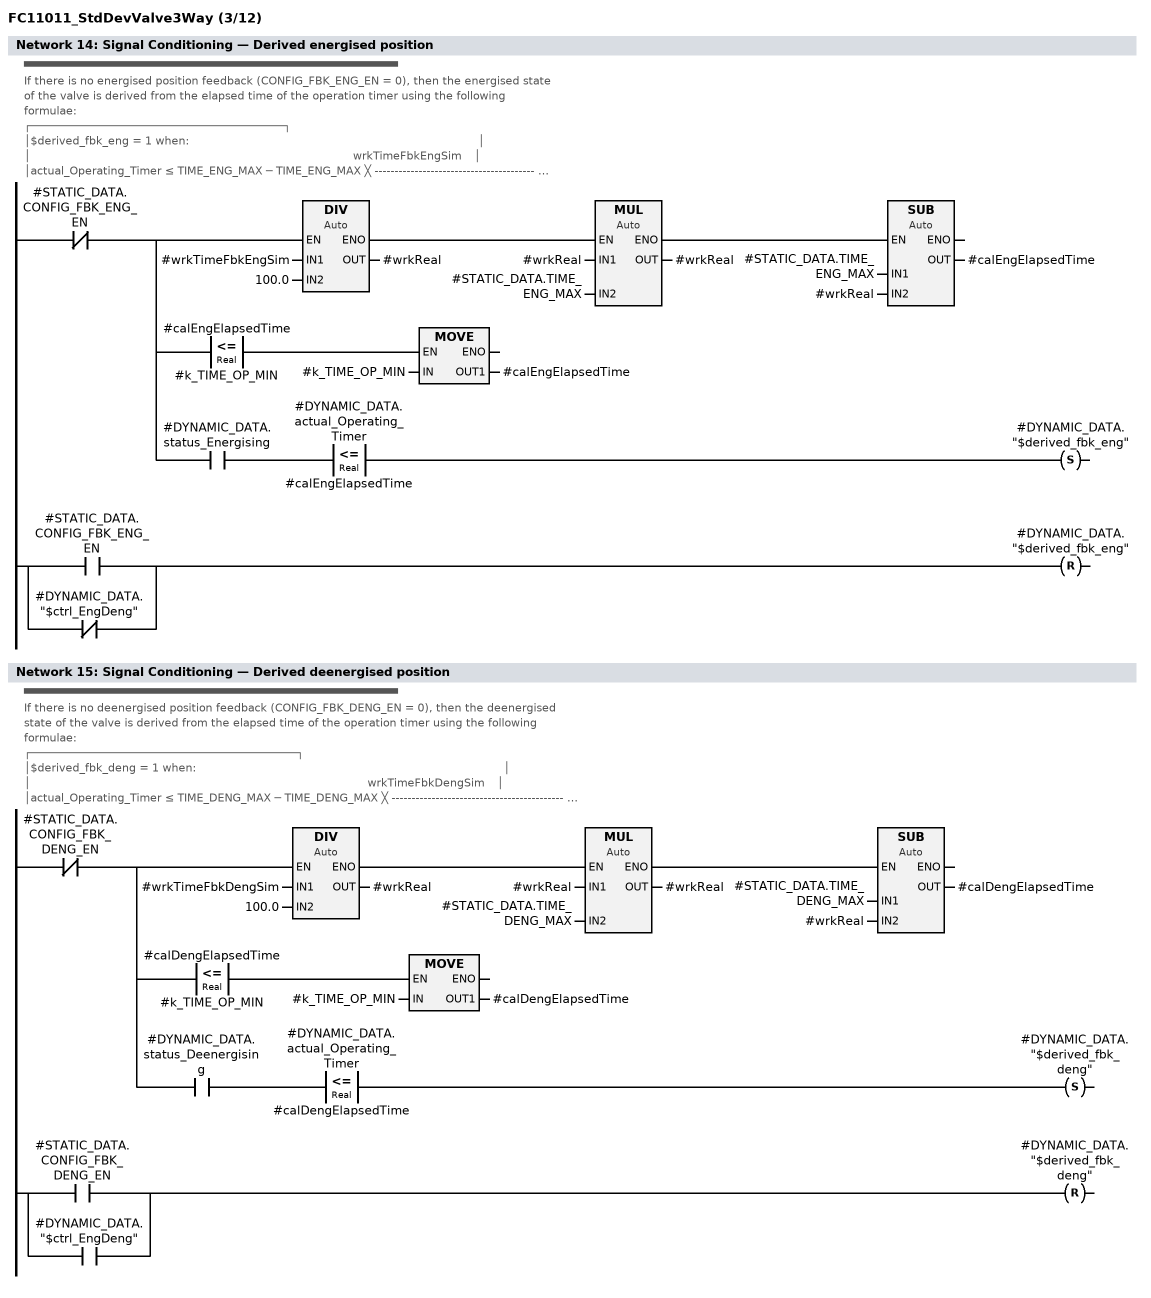
   RUNG wire#powerrail
      I_Contact( #STATIC_DATA.CONFIG_FBK_ENG_EN )
      wire#w1
      Div(in1 := #wrkTimeFbkEngSim, in2 := 100.0, out => #wrkReal)
      Mul(in1 := #wrkReal, in2 := #STATIC_DATA.TIME_ENG_MAX, out => #wrkReal)
      Sub(in1 := #STATIC_DATA.TIME_ENG_MAX, in2 := #wrkReal, out => #calEngElapsedTime)
   END_RUNG
   RUNG wire#w1
      { S7_Templates := "SrcType := Real" } LE_Contact(in1 := #calEngElapsedTime, in2 := #k_TIME_OP_MIN)
      Move(in := #k_TIME_OP_MIN, out1 => #calEngElapsedTime)
   END_RUNG
   RUNG wire#w1
      Contact( #DYNAMIC_DATA.status_Energising )
      { S7_Templates := "SrcType := Real" } LE_Contact(in1 := #DYNAMIC_DATA.actual_Operating_Timer, in2 := #calEngElapsedTime)
      S_Coil( #DYNAMIC_DATA."$derived_fbk_eng" )
   END_RUNG
   RUNG wire#powerrail
      Contact( #STATIC_DATA.CONFIG_FBK_ENG_EN )
      wire#w2
      R_Coil( #DYNAMIC_DATA."$derived_fbk_eng" )
   END_RUNG
   RUNG wire#powerrail
      I_Contact( #DYNAMIC_DATA."$ctrl_EngDeng" )
   END_RUNG wire#w2
   // the same network as SCL:
   #_w1 := NOT #STATIC_DATA.CONFIG_FBK_ENG_EN;
   IF #_w1 THEN
       #wrkReal := #wrkTimeFbkEngSim / 100.0;
       #wrkReal := #wrkReal * #STATIC_DATA.TIME_ENG_MAX;
       #calEngElapsedTime := #STATIC_DATA.TIME_ENG_MAX - #wrkReal;
   END_IF;
   IF #_w1 AND (#calEngElapsedTime <= #k_TIME_OP_MIN) THEN #calEngElapsedTime := #k_TIME_OP_MIN; END_IF;
   IF #_w1 AND #DYNAMIC_DATA.status_Energising AND (#DYNAMIC_DATA.actual_Operating_Timer <= #calEngElapsedTime) THEN
       #DYNAMIC_DATA."$derived_fbk_eng" := TRUE;
   END_IF;
   IF #STATIC_DATA.CONFIG_FBK_ENG_EN OR NOT #DYNAMIC_DATA."$ctrl_EngDeng" THEN
       #DYNAMIC_DATA."$derived_fbk_eng" := FALSE;
   END_IF;
END_REGION

REGION Network 15: Signal Conditioning — Derived deenergised position
   // ▀▀▀▀▀▀▀▀▀▀▀▀▀▀▀▀▀▀▀▀▀▀▀▀▀▀▀▀▀▀▀▀▀▀▀▀▀▀▀▀▀▀▀▀
   // If there is no deenergised position feedback (CONFIG_FBK_DENG_EN = 0), then the deenergised 
   // state of the valve is derived from the elapsed time of the operation timer using the following 
   // formulae:
   // 
   // ┌─────────────────────────────────────────┐
   // │$derived_fbk_deng = 1 when:                                 │
   // │                                wrkTimeFbkDengSim    │
   // │actual_Operating_Timer ≤ TIME_DENG_MAX ─ TIME_DENG_MAX ╳ ------------------------------------------- │
   // │                                   100           │
   // └─────────────────────────────────────────┘
   // Note:    wrkTimeFbkDengSim is the error checked equivalent of TIME_DER_DENG
   // 
   // If the calculated elapsed time is close to or less than k_TIME_OP_MIN (210ms),
   // the calculated elapsed time (calDengElapsedTime) is set to k_TIME_OP_MIN. This ensures at
   // least one timing pulse is required before the timer reaches zero.
   // 
   // The derived deenergised signal ($derived_fbk_deng) is reset if the valve is requested to be 
   // energised ($ctrl_EngDeng = 1).
   // ▄▄▄▄▄▄▄▄▄▄▄▄▄▄▄▄▄▄▄▄▄▄▄▄▄▄▄▄▄▄▄▄▄▄▄▄▄▄▄▄▄▄▄▄
   RUNG wire#powerrail
      I_Contact( #STATIC_DATA.CONFIG_FBK_DENG_EN )
      wire#w1
      Div(in1 := #wrkTimeFbkDengSim, in2 := 100.0, out => #wrkReal)
      Mul(in1 := #wrkReal, in2 := #STATIC_DATA.TIME_DENG_MAX, out => #wrkReal)
      Sub(in1 := #STATIC_DATA.TIME_DENG_MAX, in2 := #wrkReal, out => #calDengElapsedTime)
   END_RUNG
   RUNG wire#w1
      { S7_Templates := "SrcType := Real" } LE_Contact(in1 := #calDengElapsedTime, in2 := #k_TIME_OP_MIN)
      Move(in := #k_TIME_OP_MIN, out1 => #calDengElapsedTime)
   END_RUNG
   RUNG wire#w1
      Contact( #DYNAMIC_DATA.status_Deenergising )
      { S7_Templates := "SrcType := Real" } LE_Contact(in1 := #DYNAMIC_DATA.actual_Operating_Timer, in2 := #calDengElapsedTime)
      S_Coil( #DYNAMIC_DATA."$derived_fbk_deng" )
   END_RUNG
   RUNG wire#powerrail
      Contact( #STATIC_DATA.CONFIG_FBK_DENG_EN )
      wire#w2
      R_Coil( #DYNAMIC_DATA."$derived_fbk_deng" )
   END_RUNG
   RUNG wire#powerrail
      Contact( #DYNAMIC_DATA."$ctrl_EngDeng" )
   END_RUNG wire#w2
   // the same network as SCL:
   #_w1 := NOT #STATIC_DATA.CONFIG_FBK_DENG_EN;
   IF #_w1 THEN
       #wrkReal := #wrkTimeFbkDengSim / 100.0;
       #wrkReal := #wrkReal * #STATIC_DATA.TIME_DENG_MAX;
       #calDengElapsedTime := #STATIC_DATA.TIME_DENG_MAX - #wrkReal;
   END_IF;
   IF #_w1 AND (#calDengElapsedTime <= #k_TIME_OP_MIN) THEN #calDengElapsedTime := #k_TIME_OP_MIN; END_IF;
   IF #_w1 AND #DYNAMIC_DATA.status_Deenergising AND (#DYNAMIC_DATA.actual_Operating_Timer <= #calDengElapsedTime) THEN
       #DYNAMIC_DATA."$derived_fbk_deng" := TRUE;
   END_IF;
   IF #STATIC_DATA.CONFIG_FBK_DENG_EN OR #DYNAMIC_DATA."$ctrl_EngDeng" THEN
       #DYNAMIC_DATA."$derived_fbk_deng" := FALSE;
   END_IF;
END_REGION

REGION Network 16: Signal Conditioning — Simulation mode — Energised signal
   // ▀▀▀▀▀▀▀▀▀▀▀▀▀▀▀▀▀▀▀▀▀▀▀▀▀▀▀▀▀▀▀▀▀▀▀▀▀▀▀▀▀▀▀▀
   // If simulation mode is active, the simulated energised position signal is set as follows:
   // 
   //    •   mode_SimValue = 0 (no feedback), $sim_fbk_eng = 0
   // 
   //    •   mode_SimValue = 1 (permanently energised), $sim_fbk_eng = 1
   // 
   //    •   mode_SimValue = 2 (permanently deenergised), $sim_fbk_eng = 0
   // 
   //    •   mode_SimValue = 3 (follow demand), $sim_fbk_eng = $ctrl_EngDeng
   // 
   // If simulation mode is not active,  $sim_fbk_eng = 0
   // ▄▄▄▄▄▄▄▄▄▄▄▄▄▄▄▄▄▄▄▄▄▄▄▄▄▄▄▄▄▄▄▄▄▄▄▄▄▄▄▄▄▄▄▄
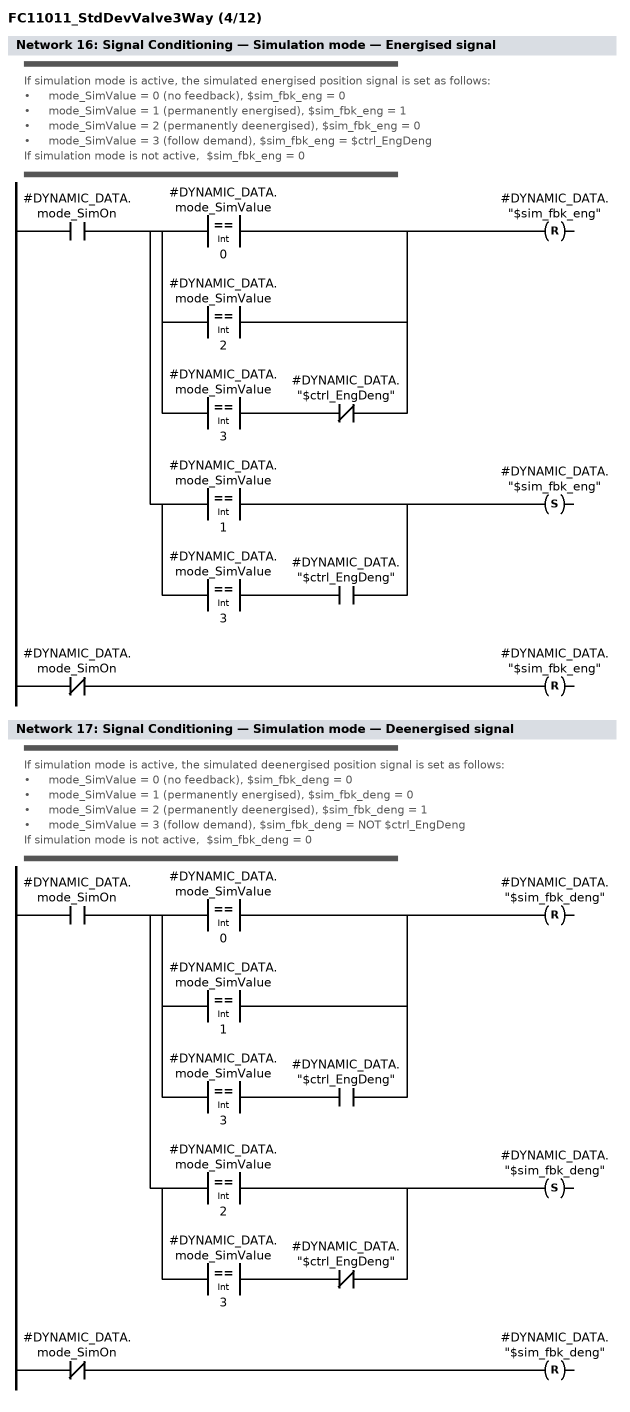
   RUNG wire#powerrail
      Contact( #DYNAMIC_DATA.mode_SimOn )
      wire#w1
      { S7_Templates := "SrcType := Int" } EQ_Contact(in1 := #DYNAMIC_DATA.mode_SimValue, in2 := 0)
      wire#w2
      R_Coil( #DYNAMIC_DATA."$sim_fbk_eng" )
   END_RUNG
   RUNG wire#w1
      { S7_Templates := "SrcType := Int" } EQ_Contact(in1 := #DYNAMIC_DATA.mode_SimValue, in2 := 2)
   END_RUNG wire#w2
   RUNG wire#w1
      { S7_Templates := "SrcType := Int" } EQ_Contact(in1 := #DYNAMIC_DATA.mode_SimValue, in2 := 3)
      I_Contact( #DYNAMIC_DATA."$ctrl_EngDeng" )
   END_RUNG wire#w2
   RUNG wire#w1
      { S7_Templates := "SrcType := Int" } EQ_Contact(in1 := #DYNAMIC_DATA.mode_SimValue, in2 := 1)
      wire#w3
      S_Coil( #DYNAMIC_DATA."$sim_fbk_eng" )
   END_RUNG
   RUNG wire#w1
      { S7_Templates := "SrcType := Int" } EQ_Contact(in1 := #DYNAMIC_DATA.mode_SimValue, in2 := 3)
      Contact( #DYNAMIC_DATA."$ctrl_EngDeng" )
   END_RUNG wire#w3
   RUNG wire#powerrail
      I_Contact( #DYNAMIC_DATA.mode_SimOn )
      R_Coil( #DYNAMIC_DATA."$sim_fbk_eng" )
   END_RUNG
   // the same network as SCL:
   IF #DYNAMIC_DATA.mode_SimOn AND ((#DYNAMIC_DATA.mode_SimValue = 0) OR (#DYNAMIC_DATA.mode_SimValue = 2) OR ((#DYNAMIC_DATA.mode_SimValue = 3) AND NOT #DYNAMIC_DATA."$ctrl_EngDeng")) THEN
       #DYNAMIC_DATA."$sim_fbk_eng" := FALSE;
   END_IF;
   IF #DYNAMIC_DATA.mode_SimOn AND ((#DYNAMIC_DATA.mode_SimValue = 1) OR ((#DYNAMIC_DATA.mode_SimValue = 3) AND #DYNAMIC_DATA."$ctrl_EngDeng")) THEN
       #DYNAMIC_DATA."$sim_fbk_eng" := TRUE;
   END_IF;
   IF NOT #DYNAMIC_DATA.mode_SimOn THEN #DYNAMIC_DATA."$sim_fbk_eng" := FALSE; END_IF;
END_REGION

REGION Network 17: Signal Conditioning — Simulation mode — Deenergised signal
   // ▀▀▀▀▀▀▀▀▀▀▀▀▀▀▀▀▀▀▀▀▀▀▀▀▀▀▀▀▀▀▀▀▀▀▀▀▀▀▀▀▀▀▀▀
   // If simulation mode is active, the simulated deenergised position signal is set as follows:
   // 
   //    •   mode_SimValue = 0 (no feedback), $sim_fbk_deng = 0
   // 
   //    •   mode_SimValue = 1 (permanently energised), $sim_fbk_deng = 0
   // 
   //    •   mode_SimValue = 2 (permanently deenergised), $sim_fbk_deng = 1
   // 
   //    •   mode_SimValue = 3 (follow demand), $sim_fbk_deng = NOT $ctrl_EngDeng
   // 
   // If simulation mode is not active,  $sim_fbk_deng = 0
   // ▄▄▄▄▄▄▄▄▄▄▄▄▄▄▄▄▄▄▄▄▄▄▄▄▄▄▄▄▄▄▄▄▄▄▄▄▄▄▄▄▄▄▄▄
   RUNG wire#powerrail
      Contact( #DYNAMIC_DATA.mode_SimOn )
      wire#w1
      { S7_Templates := "SrcType := Int" } EQ_Contact(in1 := #DYNAMIC_DATA.mode_SimValue, in2 := 0)
      wire#w2
      R_Coil( #DYNAMIC_DATA."$sim_fbk_deng" )
   END_RUNG
   RUNG wire#w1
      { S7_Templates := "SrcType := Int" } EQ_Contact(in1 := #DYNAMIC_DATA.mode_SimValue, in2 := 1)
   END_RUNG wire#w2
   RUNG wire#w1
      { S7_Templates := "SrcType := Int" } EQ_Contact(in1 := #DYNAMIC_DATA.mode_SimValue, in2 := 3)
      Contact( #DYNAMIC_DATA."$ctrl_EngDeng" )
   END_RUNG wire#w2
   RUNG wire#w1
      { S7_Templates := "SrcType := Int" } EQ_Contact(in1 := #DYNAMIC_DATA.mode_SimValue, in2 := 2)
      wire#w3
      S_Coil( #DYNAMIC_DATA."$sim_fbk_deng" )
   END_RUNG
   RUNG wire#w1
      { S7_Templates := "SrcType := Int" } EQ_Contact(in1 := #DYNAMIC_DATA.mode_SimValue, in2 := 3)
      I_Contact( #DYNAMIC_DATA."$ctrl_EngDeng" )
   END_RUNG wire#w3
   RUNG wire#powerrail
      I_Contact( #DYNAMIC_DATA.mode_SimOn )
      R_Coil( #DYNAMIC_DATA."$sim_fbk_deng" )
   END_RUNG
   // the same network as SCL:
   IF #DYNAMIC_DATA.mode_SimOn AND ((#DYNAMIC_DATA.mode_SimValue = 0) OR (#DYNAMIC_DATA.mode_SimValue = 1) OR ((#DYNAMIC_DATA.mode_SimValue = 3) AND #DYNAMIC_DATA."$ctrl_EngDeng")) THEN
       #DYNAMIC_DATA."$sim_fbk_deng" := FALSE;
   END_IF;
   IF #DYNAMIC_DATA.mode_SimOn AND ((#DYNAMIC_DATA.mode_SimValue = 2) OR ((#DYNAMIC_DATA.mode_SimValue = 3) AND NOT #DYNAMIC_DATA."$ctrl_EngDeng")) THEN
       #DYNAMIC_DATA."$sim_fbk_deng" := TRUE;
   END_IF;
   IF NOT #DYNAMIC_DATA.mode_SimOn THEN #DYNAMIC_DATA."$sim_fbk_deng" := FALSE; END_IF;
END_REGION

REGION Network 18: Signal conditioning — Determine valve ENG position status
   // ▀▀▀▀▀▀▀▀▀▀▀▀▀▀▀▀▀▀▀▀▀▀▀▀▀▀▀▀▀▀▀▀▀▀▀▀▀▀▀▀▀▀▀▀
   // Generates a working energised signal (wrkEng), that is then used throughout the module as the 
   // definitive energised position feedback signal.
   // 
   // The energised signal will be either :
   // 
   //    1.  The same as the FBK_ENG parameter if this is in use 
   //      (CONFIG_FBK_ENG_EN = 1)
   // 
   //    2.  The internally derived energised state (based on the requested state of the valve) 
   //      if the FBK_ENG signal is NOT in use (CONFIG_FBK_ENG_EN = 0)
   // 
   //    3.  The simulated state of the valve if simulation mode is active (mode_SimOn = 1)
   // 
   // If an actual energised position signal is provided to the module via the FBK_ENG parameter 
   // (i.e. if CONFIG_FBK_ENG_EN = 1) then wrkEng is set to match the FBK_ENG signal 
   // (wrkEng = FBK_ENG).
   // 
   // If a derived energised signal is to be used (i.e. if CONFIG_FBK_ENG_EN = 0), then wrkEng is set to 
   // match the internally derived $derived_fbk_eng signal (wrkEng = $derived_fbk_eng). 
   // $derived_fbk_eng is based on the requested state of the valve. 
   // 
   // Finally, if simulation mode is active (mode_SimOn = 1), then wrkEng is set to match the internal 
   // simulation signal $sim_fbk_eng signal (wrkEng = $sim_fbk_eng).
   // ▄▄▄▄▄▄▄▄▄▄▄▄▄▄▄▄▄▄▄▄▄▄▄▄▄▄▄▄▄▄▄▄▄▄▄▄▄▄▄▄▄▄▄▄
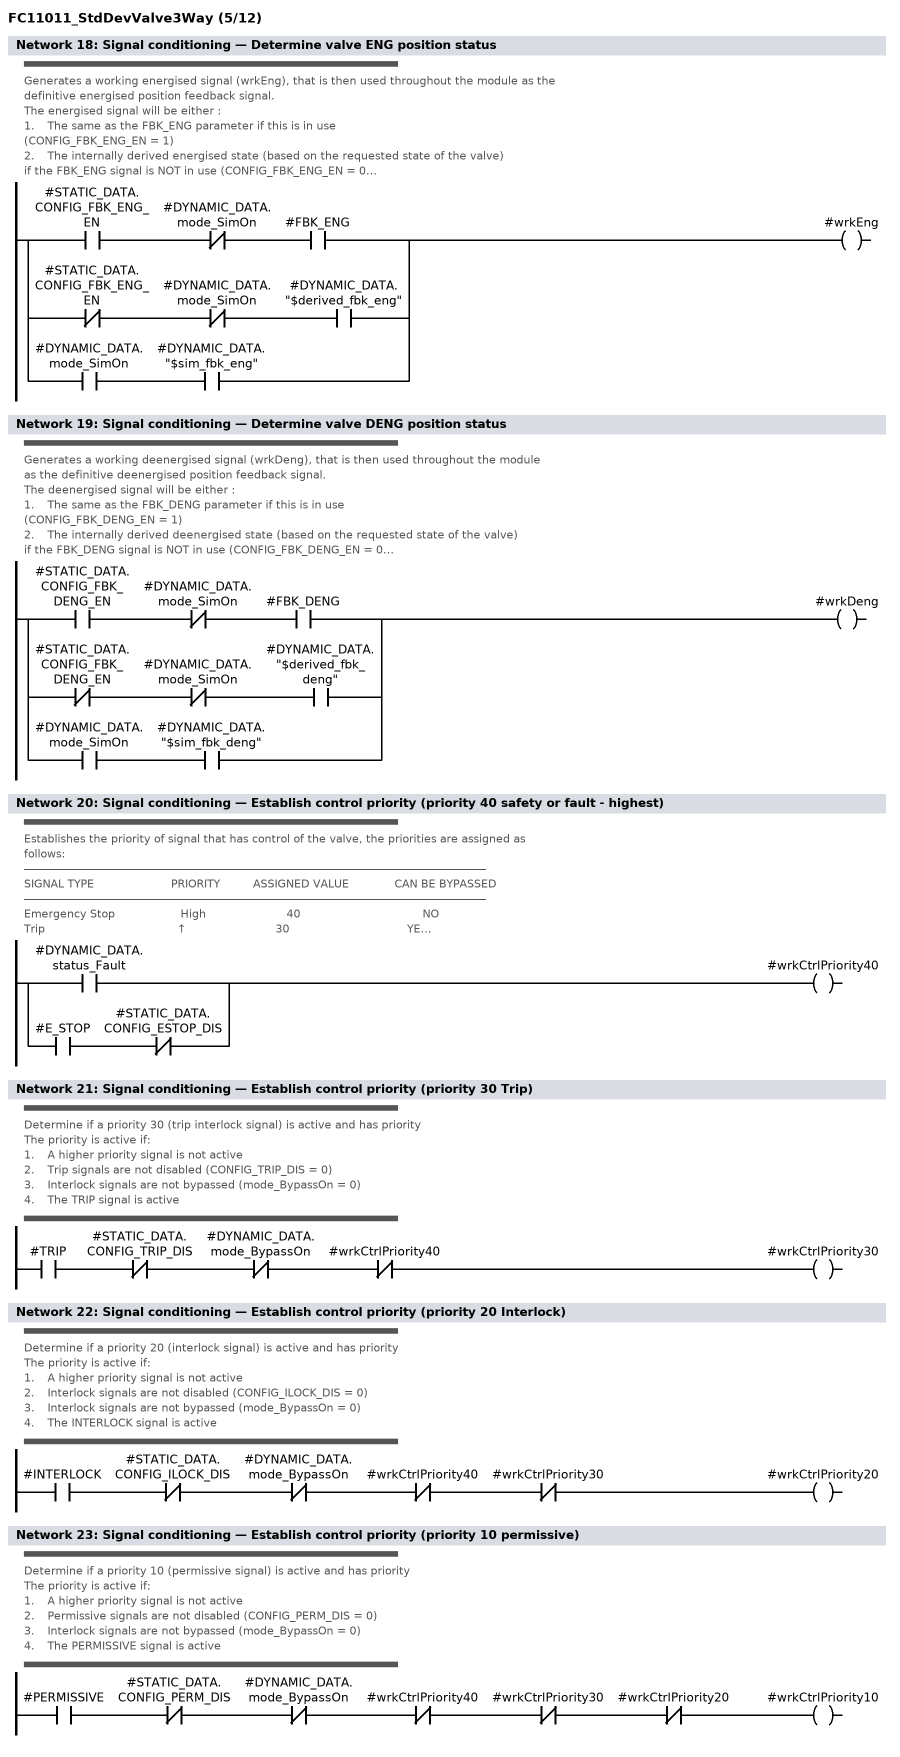
   RUNG wire#powerrail
      Contact( #STATIC_DATA.CONFIG_FBK_ENG_EN )
      I_Contact( #DYNAMIC_DATA.mode_SimOn )
      Contact( #FBK_ENG )
      wire#w1
      Coil( #wrkEng )
   END_RUNG
   RUNG wire#powerrail
      I_Contact( #STATIC_DATA.CONFIG_FBK_ENG_EN )
      I_Contact( #DYNAMIC_DATA.mode_SimOn )
      Contact( #DYNAMIC_DATA."$derived_fbk_eng" )
   END_RUNG wire#w1
   RUNG wire#powerrail
      Contact( #DYNAMIC_DATA.mode_SimOn )
      Contact( #DYNAMIC_DATA."$sim_fbk_eng" )
   END_RUNG wire#w1
   // the same network as SCL:
   #wrkEng := (#STATIC_DATA.CONFIG_FBK_ENG_EN AND NOT #DYNAMIC_DATA.mode_SimOn AND #FBK_ENG) OR (NOT #STATIC_DATA.CONFIG_FBK_ENG_EN AND NOT #DYNAMIC_DATA.mode_SimOn AND #DYNAMIC_DATA."$derived_fbk_eng") OR (#DYNAMIC_DATA.mode_SimOn AND #DYNAMIC_DATA."$sim_fbk_eng");
END_REGION

REGION Network 19: Signal conditioning — Determine valve DENG position status
   // ▀▀▀▀▀▀▀▀▀▀▀▀▀▀▀▀▀▀▀▀▀▀▀▀▀▀▀▀▀▀▀▀▀▀▀▀▀▀▀▀▀▀▀▀
   // Generates a working deenergised signal (wrkDeng), that is then used throughout the module 
   // as the definitive deenergised position feedback signal.
   // 
   // The deenergised signal will be either :
   // 
   //    1.  The same as the FBK_DENG parameter if this is in use 
   //      (CONFIG_FBK_DENG_EN = 1)
   // 
   //    2.  The internally derived deenergised state (based on the requested state of the valve) 
   //      if the FBK_DENG signal is NOT in use (CONFIG_FBK_DENG_EN = 0)
   // 
   //    3.  The simulated state of the valve if simulation mode is active (mode_SimOn = 1)
   // 
   // If an actual deenergised position signal is provided to the module via the FBK_DENG parameter 
   // (i.e. if CONFIG_FBK_DENG_EN = 1) then wrkDeng is set to match the FBK_DENG signal 
   // wrkDeng = FBK_DENG).
   // 
   // If a derived deenergised signal is to be used (i.e. if CONFIG_FBK_DENG_EN = 0), then wrkDeng is 
   // set to match the internally derived $derived_fbk_deng signal 
   // (wrkDeng = $derived_fbk_deng). $derived_fbk_deng is based on the requested state of 
   // the valve.
   // 
   // Finally, if simulation mode is active (mode_SimOn = 1), then wrkDeng is set to match the 
   // internal simulation signal $sim_fbk_deng signal (wrkDeng = $sim_fbk_deng). 
   // ▄▄▄▄▄▄▄▄▄▄▄▄▄▄▄▄▄▄▄▄▄▄▄▄▄▄▄▄▄▄▄▄▄▄▄▄▄▄▄▄▄▄▄▄
   RUNG wire#powerrail
      Contact( #STATIC_DATA.CONFIG_FBK_DENG_EN )
      I_Contact( #DYNAMIC_DATA.mode_SimOn )
      Contact( #FBK_DENG )
      wire#w1
      Coil( #wrkDeng )
   END_RUNG
   RUNG wire#powerrail
      I_Contact( #STATIC_DATA.CONFIG_FBK_DENG_EN )
      I_Contact( #DYNAMIC_DATA.mode_SimOn )
      Contact( #DYNAMIC_DATA."$derived_fbk_deng" )
   END_RUNG wire#w1
   RUNG wire#powerrail
      Contact( #DYNAMIC_DATA.mode_SimOn )
      Contact( #DYNAMIC_DATA."$sim_fbk_deng" )
   END_RUNG wire#w1
   // the same network as SCL:
   #wrkDeng := (#STATIC_DATA.CONFIG_FBK_DENG_EN AND NOT #DYNAMIC_DATA.mode_SimOn AND #FBK_DENG) OR (NOT #STATIC_DATA.CONFIG_FBK_DENG_EN AND NOT #DYNAMIC_DATA.mode_SimOn AND #DYNAMIC_DATA."$derived_fbk_deng") OR (#DYNAMIC_DATA.mode_SimOn AND #DYNAMIC_DATA."$sim_fbk_deng");
END_REGION

REGION Network 20: Signal conditioning — Establish control priority (priority 40 safety or fault - highest)
   // ▀▀▀▀▀▀▀▀▀▀▀▀▀▀▀▀▀▀▀▀▀▀▀▀▀▀▀▀▀▀▀▀▀▀▀▀▀▀▀▀▀▀▀▀
   // Establishes the priority of signal that has control of the valve, the priorities are assigned as 
   // follows:
   // 
   //  ――――――――――――――――――――――――――――――――――――――――――
   //  SIGNAL TYPE       PRIORITY   ASSIGNED VALUE       CAN BE BYPASSED
   //  ――――――――――――――――――――――――――――――――――――――――――
   //  Emergency Stop        High        40                NO
   //  Trip            ↑           30             YES
   //  Interlock            ↑           20             YES
   //  Permissive          ↑           10             YES
   //  Auto/manual control    Low         00                NO
   //  ――――――――――――――――――――――――――――――――――――――――――
   //  High priority signal take precedence over lower priority signals.
   // 
   // Determine a priority 40 (valve safety (or fault) condition is active)
   // 
   // The priority is active if:
   // 
   //    1.  The valve is in a fault condition (status_Fault = 1)
   // 
   //   OR both the following are true
   // 
   //    1.  Safety signals are not disabled (CONFIG_ESTOP_DIS = 0)
   // 
   //    2.  The E_STOP signal is active
   // ▄▄▄▄▄▄▄▄▄▄▄▄▄▄▄▄▄▄▄▄▄▄▄▄▄▄▄▄▄▄▄▄▄▄▄▄▄▄▄▄▄▄▄▄
   RUNG wire#powerrail
      Contact( #DYNAMIC_DATA.status_Fault )
      wire#w1
      Coil( #wrkCtrlPriority40 )
   END_RUNG
   RUNG wire#powerrail
      Contact( #E_STOP )
      I_Contact( #STATIC_DATA.CONFIG_ESTOP_DIS )
   END_RUNG wire#w1
   // the same network as SCL:
   #wrkCtrlPriority40 := #DYNAMIC_DATA.status_Fault OR (#E_STOP AND NOT #STATIC_DATA.CONFIG_ESTOP_DIS);
END_REGION

REGION Network 21: Signal conditioning — Establish control priority (priority 30 Trip)
   // ▀▀▀▀▀▀▀▀▀▀▀▀▀▀▀▀▀▀▀▀▀▀▀▀▀▀▀▀▀▀▀▀▀▀▀▀▀▀▀▀▀▀▀▀
   // Determine if a priority 30 (trip interlock signal) is active and has priority
   // 
   // The priority is active if:
   // 
   //    1.  A higher priority signal is not active
   // 
   //    2.  Trip signals are not disabled (CONFIG_TRIP_DIS = 0)
   // 
   //    3.  Interlock signals are not bypassed (mode_BypassOn = 0)
   // 
   //    4.  The TRIP signal is active
   // ▄▄▄▄▄▄▄▄▄▄▄▄▄▄▄▄▄▄▄▄▄▄▄▄▄▄▄▄▄▄▄▄▄▄▄▄▄▄▄▄▄▄▄▄
   RUNG wire#powerrail
      Contact( #TRIP )
      I_Contact( #STATIC_DATA.CONFIG_TRIP_DIS )
      I_Contact( #DYNAMIC_DATA.mode_BypassOn )
      I_Contact( #wrkCtrlPriority40 )
      Coil( #wrkCtrlPriority30 )
   END_RUNG
   // the same network as SCL:
   #wrkCtrlPriority30 := #TRIP AND NOT #STATIC_DATA.CONFIG_TRIP_DIS AND NOT #DYNAMIC_DATA.mode_BypassOn AND NOT #wrkCtrlPriority40;
END_REGION

REGION Network 22: Signal conditioning — Establish control priority (priority 20 Interlock)
   // ▀▀▀▀▀▀▀▀▀▀▀▀▀▀▀▀▀▀▀▀▀▀▀▀▀▀▀▀▀▀▀▀▀▀▀▀▀▀▀▀▀▀▀▀
   // Determine if a priority 20 (interlock signal) is active and has priority
   // 
   // The priority is active if:
   // 
   //    1.  A higher priority signal is not active
   // 
   //    2.  Interlock signals are not disabled (CONFIG_ILOCK_DIS = 0)
   // 
   //    3.  Interlock signals are not bypassed (mode_BypassOn = 0)
   // 
   //    4.  The INTERLOCK signal is active
   // ▄▄▄▄▄▄▄▄▄▄▄▄▄▄▄▄▄▄▄▄▄▄▄▄▄▄▄▄▄▄▄▄▄▄▄▄▄▄▄▄▄▄▄▄
   RUNG wire#powerrail
      Contact( #INTERLOCK )
      I_Contact( #STATIC_DATA.CONFIG_ILOCK_DIS )
      I_Contact( #DYNAMIC_DATA.mode_BypassOn )
      I_Contact( #wrkCtrlPriority40 )
      I_Contact( #wrkCtrlPriority30 )
      Coil( #wrkCtrlPriority20 )
   END_RUNG
   // the same network as SCL:
   #wrkCtrlPriority20 := #INTERLOCK AND NOT #STATIC_DATA.CONFIG_ILOCK_DIS AND NOT #DYNAMIC_DATA.mode_BypassOn AND NOT #wrkCtrlPriority40 AND NOT #wrkCtrlPriority30;
END_REGION

REGION Network 23: Signal conditioning — Establish control priority (priority 10 permissive)
   // ▀▀▀▀▀▀▀▀▀▀▀▀▀▀▀▀▀▀▀▀▀▀▀▀▀▀▀▀▀▀▀▀▀▀▀▀▀▀▀▀▀▀▀▀
   // Determine if a priority 10 (permissive signal) is active and has priority
   // 
   // The priority is active if:
   // 
   //    1.  A higher priority signal is not active
   // 
   //    2.  Permissive signals are not disabled (CONFIG_PERM_DIS = 0)
   // 
   //    3.  Interlock signals are not bypassed (mode_BypassOn = 0)
   // 
   //    4.  The PERMISSIVE signal is active
   // ▄▄▄▄▄▄▄▄▄▄▄▄▄▄▄▄▄▄▄▄▄▄▄▄▄▄▄▄▄▄▄▄▄▄▄▄▄▄▄▄▄▄▄▄
   RUNG wire#powerrail
      Contact( #PERMISSIVE )
      I_Contact( #STATIC_DATA.CONFIG_PERM_DIS )
      I_Contact( #DYNAMIC_DATA.mode_BypassOn )
      I_Contact( #wrkCtrlPriority40 )
      I_Contact( #wrkCtrlPriority30 )
      I_Contact( #wrkCtrlPriority20 )
      Coil( #wrkCtrlPriority10 )
   END_RUNG
   // the same network as SCL:
   #wrkCtrlPriority10 := #PERMISSIVE AND NOT #STATIC_DATA.CONFIG_PERM_DIS AND NOT #DYNAMIC_DATA.mode_BypassOn AND NOT #wrkCtrlPriority40 AND NOT #wrkCtrlPriority30 AND NOT #wrkCtrlPriority20;
END_REGION

REGION Network 24: Signal conditioning — Establish control priority (priority 00 auto/manual - lowest)
   // ▀▀▀▀▀▀▀▀▀▀▀▀▀▀▀▀▀▀▀▀▀▀▀▀▀▀▀▀▀▀▀▀▀▀▀▀▀▀▀▀▀▀▀▀
   // Determine if a priority 00 (automatic or manual control) is active and has priority
   // 
   // The priority is active if:
   // 
   //    1.  A higher priority signal is not active
   // ▄▄▄▄▄▄▄▄▄▄▄▄▄▄▄▄▄▄▄▄▄▄▄▄▄▄▄▄▄▄▄▄▄▄▄▄▄▄▄▄▄▄▄▄
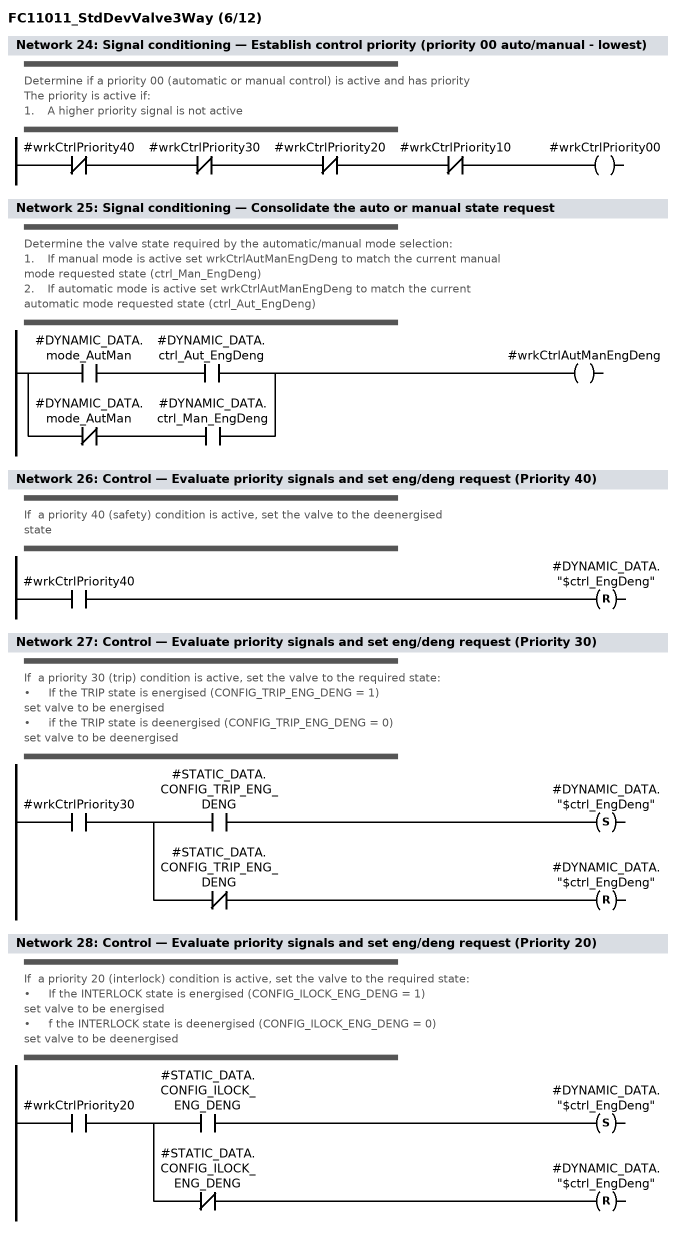
   RUNG wire#powerrail
      I_Contact( #wrkCtrlPriority40 )
      I_Contact( #wrkCtrlPriority30 )
      I_Contact( #wrkCtrlPriority20 )
      I_Contact( #wrkCtrlPriority10 )
      Coil( #wrkCtrlPriority00 )
   END_RUNG
   // the same network as SCL:
   #wrkCtrlPriority00 := NOT #wrkCtrlPriority40 AND NOT #wrkCtrlPriority30 AND NOT #wrkCtrlPriority20 AND NOT #wrkCtrlPriority10;
END_REGION

REGION Network 25: Signal conditioning — Consolidate the auto or manual state request
   // ▀▀▀▀▀▀▀▀▀▀▀▀▀▀▀▀▀▀▀▀▀▀▀▀▀▀▀▀▀▀▀▀▀▀▀▀▀▀▀▀▀▀▀▀
   // Determine the valve state required by the automatic/manual mode selection:
   // 
   //    1.  If manual mode is active set wrkCtrlAutManEngDeng to match the current manual 
   //      mode requested state (ctrl_Man_EngDeng)
   // 
   //    2.  If automatic mode is active set wrkCtrlAutManEngDeng to match the current 
   //      automatic mode requested state (ctrl_Aut_EngDeng)
   // ▄▄▄▄▄▄▄▄▄▄▄▄▄▄▄▄▄▄▄▄▄▄▄▄▄▄▄▄▄▄▄▄▄▄▄▄▄▄▄▄▄▄▄▄
   RUNG wire#powerrail
      Contact( #DYNAMIC_DATA.mode_AutMan )
      Contact( #DYNAMIC_DATA.ctrl_Aut_EngDeng )
      wire#w1
      Coil( #wrkCtrlAutManEngDeng )
   END_RUNG
   RUNG wire#powerrail
      I_Contact( #DYNAMIC_DATA.mode_AutMan )
      Contact( #DYNAMIC_DATA.ctrl_Man_EngDeng )
   END_RUNG wire#w1
   // the same network as SCL:
   #wrkCtrlAutManEngDeng := (#DYNAMIC_DATA.mode_AutMan AND #DYNAMIC_DATA.ctrl_Aut_EngDeng) OR (NOT #DYNAMIC_DATA.mode_AutMan AND #DYNAMIC_DATA.ctrl_Man_EngDeng);
END_REGION

REGION Network 26: Control — Evaluate priority signals and set eng/deng request (Priority 40)
   // ▀▀▀▀▀▀▀▀▀▀▀▀▀▀▀▀▀▀▀▀▀▀▀▀▀▀▀▀▀▀▀▀▀▀▀▀▀▀▀▀▀▀▀▀
   // If  a priority 40 (safety) condition is active, set the valve to the deenergised 
   // state
   // ▄▄▄▄▄▄▄▄▄▄▄▄▄▄▄▄▄▄▄▄▄▄▄▄▄▄▄▄▄▄▄▄▄▄▄▄▄▄▄▄▄▄▄▄
   RUNG wire#powerrail
      Contact( #wrkCtrlPriority40 )
      R_Coil( #DYNAMIC_DATA."$ctrl_EngDeng" )
   END_RUNG
   // the same network as SCL:
   IF #wrkCtrlPriority40 THEN #DYNAMIC_DATA."$ctrl_EngDeng" := FALSE; END_IF;
END_REGION

REGION Network 27: Control — Evaluate priority signals and set eng/deng request (Priority 30)
   // ▀▀▀▀▀▀▀▀▀▀▀▀▀▀▀▀▀▀▀▀▀▀▀▀▀▀▀▀▀▀▀▀▀▀▀▀▀▀▀▀▀▀▀▀
   // If  a priority 30 (trip) condition is active, set the valve to the required state:
   // 
   //    •   If the TRIP state is energised (CONFIG_TRIP_ENG_DENG = 1) 
   //      set valve to be energised
   // 
   //    •   if the TRIP state is deenergised (CONFIG_TRIP_ENG_DENG = 0) 
   //      set valve to be deenergised
   // ▄▄▄▄▄▄▄▄▄▄▄▄▄▄▄▄▄▄▄▄▄▄▄▄▄▄▄▄▄▄▄▄▄▄▄▄▄▄▄▄▄▄▄▄
   RUNG wire#powerrail
      Contact( #wrkCtrlPriority30 )
      wire#w1
      Contact( #STATIC_DATA.CONFIG_TRIP_ENG_DENG )
      S_Coil( #DYNAMIC_DATA."$ctrl_EngDeng" )
   END_RUNG
   RUNG wire#w1
      I_Contact( #STATIC_DATA.CONFIG_TRIP_ENG_DENG )
      R_Coil( #DYNAMIC_DATA."$ctrl_EngDeng" )
   END_RUNG
   // the same network as SCL:
   IF #wrkCtrlPriority30 AND #STATIC_DATA.CONFIG_TRIP_ENG_DENG THEN
       #DYNAMIC_DATA."$ctrl_EngDeng" := TRUE;
   END_IF;
   IF #wrkCtrlPriority30 AND NOT #STATIC_DATA.CONFIG_TRIP_ENG_DENG THEN
       #DYNAMIC_DATA."$ctrl_EngDeng" := FALSE;
   END_IF;
END_REGION

REGION Network 28: Control — Evaluate priority signals and set eng/deng request (Priority 20)
   // ▀▀▀▀▀▀▀▀▀▀▀▀▀▀▀▀▀▀▀▀▀▀▀▀▀▀▀▀▀▀▀▀▀▀▀▀▀▀▀▀▀▀▀▀
   // If  a priority 20 (interlock) condition is active, set the valve to the required state:
   // 
   //    •   If the INTERLOCK state is energised (CONFIG_ILOCK_ENG_DENG = 1) 
   //      set valve to be energised
   // 
   //    •   f the INTERLOCK state is deenergised (CONFIG_ILOCK_ENG_DENG = 0) 
   //      set valve to be deenergised
   // ▄▄▄▄▄▄▄▄▄▄▄▄▄▄▄▄▄▄▄▄▄▄▄▄▄▄▄▄▄▄▄▄▄▄▄▄▄▄▄▄▄▄▄▄
   RUNG wire#powerrail
      Contact( #wrkCtrlPriority20 )
      wire#w1
      Contact( #STATIC_DATA.CONFIG_ILOCK_ENG_DENG )
      S_Coil( #DYNAMIC_DATA."$ctrl_EngDeng" )
   END_RUNG
   RUNG wire#w1
      I_Contact( #STATIC_DATA.CONFIG_ILOCK_ENG_DENG )
      R_Coil( #DYNAMIC_DATA."$ctrl_EngDeng" )
   END_RUNG
   // the same network as SCL:
   IF #wrkCtrlPriority20 AND #STATIC_DATA.CONFIG_ILOCK_ENG_DENG THEN
       #DYNAMIC_DATA."$ctrl_EngDeng" := TRUE;
   END_IF;
   IF #wrkCtrlPriority20 AND NOT #STATIC_DATA.CONFIG_ILOCK_ENG_DENG THEN
       #DYNAMIC_DATA."$ctrl_EngDeng" := FALSE;
   END_IF;
END_REGION

REGION Network 29: Control — Evaluate priority signals and set eng/deng request (Priority 10)
   // ▀▀▀▀▀▀▀▀▀▀▀▀▀▀▀▀▀▀▀▀▀▀▀▀▀▀▀▀▀▀▀▀▀▀▀▀▀▀▀▀▀▀▀▀
   // If  a priority 10 (permissive) condition is active, set the valve to the required state:
   // 
   // 
   // PERMITTED STATE IS ENERGISED — CONDITIONS:
   // 
   //    •   If the Permitted state is energised and Aut/Man request is for energised
   //      set the valve to be energised[Branch 1]
   // 
   //    •   If the Permitted state is energised and Aut/Man request is for deenergised and the 
   //      current valve output matches this state (deenergised) set the valve to be 
   //      deenergised (maintain the current state) [Branch 6]
   // 
   //    •   If the Permitted state is energised and Aut/Man request is for deenergised and the 
   //      current valve output matches the deenergised state, set the valve to be energised 
   //      (override the auto/man request [Branch 2]
   // 
   // PERMITTED STATE IS DEENERGISED — CONDITIONS:
   // 
   //    •   If the Permitted state is deenergised and Aut/Man request is for deenergised,
   //      set the valve to be  deenergised [Branch 4]
   // 
   //    •   If the Permitted state is deenergised and Aut/Man request is for energised, and the 
   //      current valve output matches this state (energised) set the valve to be energised 
   //      (maintain the current state) [Branch 3]
   // 
   //    •   If the Permitted state is deenergised and Aut/Man request is for energised, and the current
   //      valve output matches the deenergised  state, set the valve to be deenergised 
   //      (override the auto/man request [Branch 5]
   // ▄▄▄▄▄▄▄▄▄▄▄▄▄▄▄▄▄▄▄▄▄▄▄▄▄▄▄▄▄▄▄▄▄▄▄▄▄▄▄▄▄▄▄▄
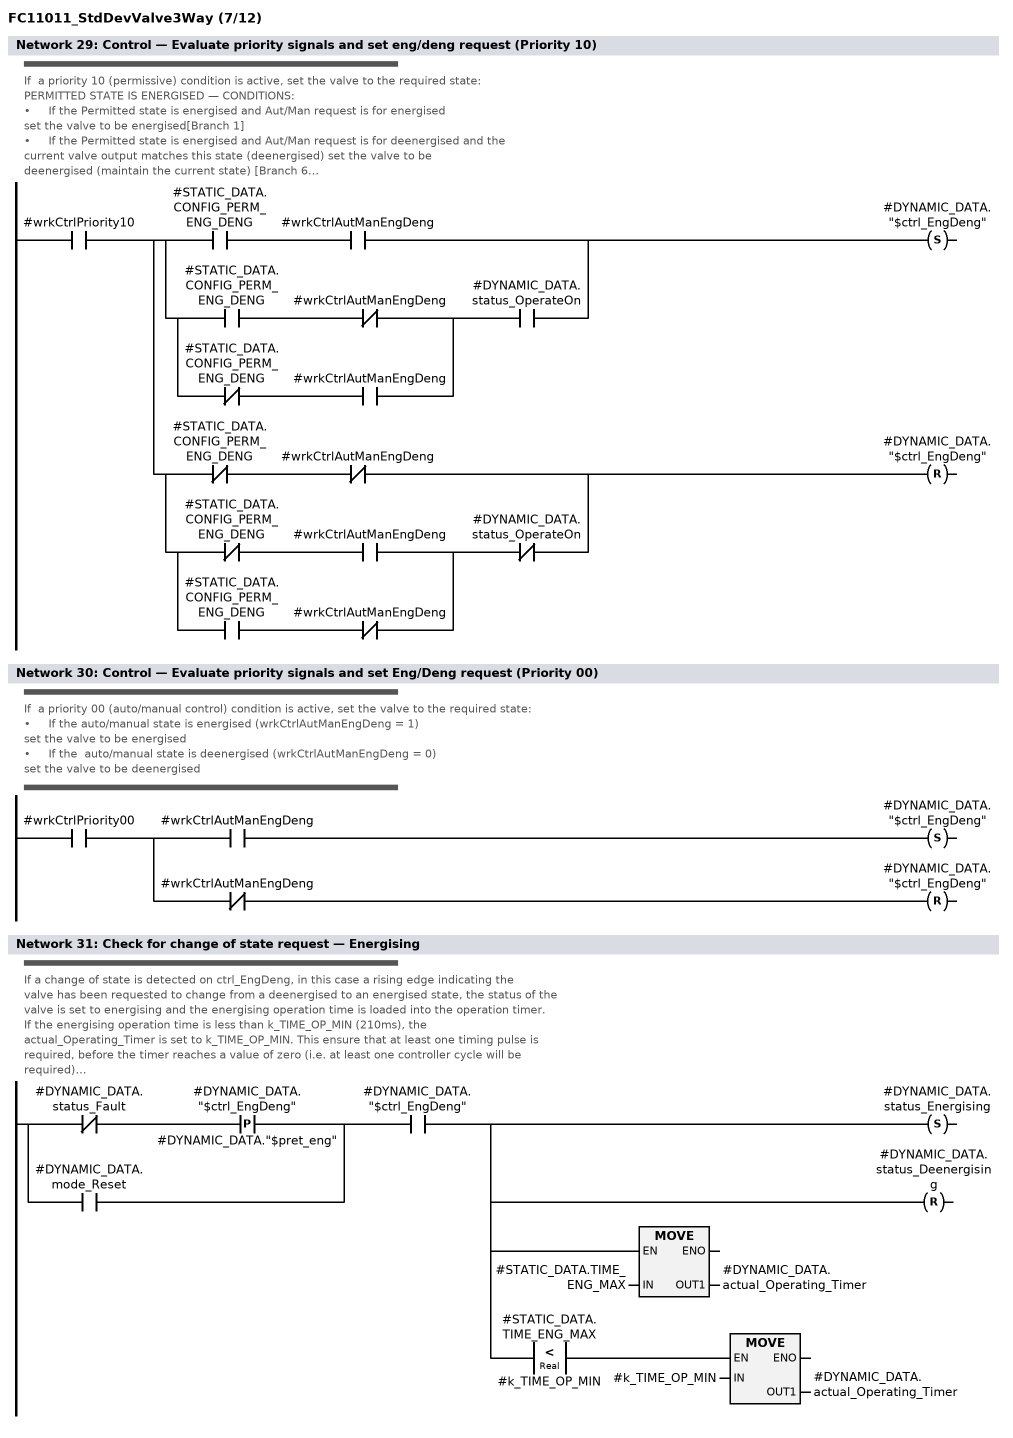
   RUNG wire#powerrail
      Contact( #wrkCtrlPriority10 )
      wire#w1
      Contact( #STATIC_DATA.CONFIG_PERM_ENG_DENG )
      Contact( #wrkCtrlAutManEngDeng )
      wire#w2
      S_Coil( #DYNAMIC_DATA."$ctrl_EngDeng" )
   END_RUNG
   RUNG wire#w1
      Contact( #STATIC_DATA.CONFIG_PERM_ENG_DENG )
      I_Contact( #wrkCtrlAutManEngDeng )
      wire#w3
      Contact( #DYNAMIC_DATA.status_OperateOn )
   END_RUNG wire#w2
   RUNG wire#w1
      I_Contact( #STATIC_DATA.CONFIG_PERM_ENG_DENG )
      Contact( #wrkCtrlAutManEngDeng )
   END_RUNG wire#w3
   RUNG wire#w1
      I_Contact( #STATIC_DATA.CONFIG_PERM_ENG_DENG )
      I_Contact( #wrkCtrlAutManEngDeng )
      wire#w4
      R_Coil( #DYNAMIC_DATA."$ctrl_EngDeng" )
   END_RUNG
   RUNG wire#w1
      I_Contact( #STATIC_DATA.CONFIG_PERM_ENG_DENG )
      Contact( #wrkCtrlAutManEngDeng )
      wire#w5
      I_Contact( #DYNAMIC_DATA.status_OperateOn )
   END_RUNG wire#w4
   RUNG wire#w1
      Contact( #STATIC_DATA.CONFIG_PERM_ENG_DENG )
      I_Contact( #wrkCtrlAutManEngDeng )
   END_RUNG wire#w5
   // the same network as SCL:
   IF #wrkCtrlPriority10 AND ((#STATIC_DATA.CONFIG_PERM_ENG_DENG AND #wrkCtrlAutManEngDeng) OR (((#STATIC_DATA.CONFIG_PERM_ENG_DENG AND NOT #wrkCtrlAutManEngDeng) OR (NOT #STATIC_DATA.CONFIG_PERM_ENG_DENG AND #wrkCtrlAutManEngDeng)) AND #DYNAMIC_DATA.status_OperateOn)) THEN
       #DYNAMIC_DATA."$ctrl_EngDeng" := TRUE;
   END_IF;
   IF #wrkCtrlPriority10 AND ((NOT #STATIC_DATA.CONFIG_PERM_ENG_DENG AND NOT #wrkCtrlAutManEngDeng) OR (((NOT #STATIC_DATA.CONFIG_PERM_ENG_DENG AND #wrkCtrlAutManEngDeng) OR (#STATIC_DATA.CONFIG_PERM_ENG_DENG AND NOT #wrkCtrlAutManEngDeng)) AND NOT #DYNAMIC_DATA.status_OperateOn)) THEN
       #DYNAMIC_DATA."$ctrl_EngDeng" := FALSE;
   END_IF;
END_REGION

REGION Network 30: Control — Evaluate priority signals and set Eng/Deng request (Priority 00)
   // ▀▀▀▀▀▀▀▀▀▀▀▀▀▀▀▀▀▀▀▀▀▀▀▀▀▀▀▀▀▀▀▀▀▀▀▀▀▀▀▀▀▀▀▀
   // If  a priority 00 (auto/manual control) condition is active, set the valve to the required state:
   // 
   //    •   If the auto/manual state is energised (wrkCtrlAutManEngDeng = 1) 
   //      set the valve to be energised
   // 
   //    •   If the  auto/manual state is deenergised (wrkCtrlAutManEngDeng = 0) 
   //      set the valve to be deenergised
   // ▄▄▄▄▄▄▄▄▄▄▄▄▄▄▄▄▄▄▄▄▄▄▄▄▄▄▄▄▄▄▄▄▄▄▄▄▄▄▄▄▄▄▄▄
   RUNG wire#powerrail
      Contact( #wrkCtrlPriority00 )
      wire#w1
      Contact( #wrkCtrlAutManEngDeng )
      S_Coil( #DYNAMIC_DATA."$ctrl_EngDeng" )
   END_RUNG
   RUNG wire#w1
      I_Contact( #wrkCtrlAutManEngDeng )
      R_Coil( #DYNAMIC_DATA."$ctrl_EngDeng" )
   END_RUNG
   // the same network as SCL:
   IF #wrkCtrlPriority00 AND #wrkCtrlAutManEngDeng THEN #DYNAMIC_DATA."$ctrl_EngDeng" := TRUE; END_IF;
   IF #wrkCtrlPriority00 AND NOT #wrkCtrlAutManEngDeng THEN #DYNAMIC_DATA."$ctrl_EngDeng" := FALSE; END_IF;
END_REGION

REGION Network 31: Check for change of state request — Energising
   // ▀▀▀▀▀▀▀▀▀▀▀▀▀▀▀▀▀▀▀▀▀▀▀▀▀▀▀▀▀▀▀▀▀▀▀▀▀▀▀▀▀▀▀▀
   // If a change of state is detected on ctrl_EngDeng, in this case a rising edge indicating the
   // valve has been requested to change from a deenergised to an energised state, the status of the
   // valve is set to energising and the energising operation time is loaded into the operation timer.
   // 
   // If the energising operation time is less than k_TIME_OP_MIN (210ms), the 
   // actual_Operating_Timer is set to k_TIME_OP_MIN. This ensure that at least one timing pulse is 
   // required, before the timer reaches a value of zero (i.e. at least one controller cycle will be 
   // required).
   // 
   // If the valve is in a fault condition (status_Fault = true), the change of state is not evaluated
   // until the fault condition has cleared
   // 
   // Note: the timer is also triggered if the Reset signal is received and the valve is requested to be 
   //            energised
   // ▄▄▄▄▄▄▄▄▄▄▄▄▄▄▄▄▄▄▄▄▄▄▄▄▄▄▄▄▄▄▄▄▄▄▄▄▄▄▄▄▄▄▄▄
   RUNG wire#powerrail
      I_Contact( #DYNAMIC_DATA.status_Fault )
      P_Contact(operand := #DYNAMIC_DATA."$ctrl_EngDeng", bit := #DYNAMIC_DATA."$pret_eng")
      wire#w1
      Contact( #DYNAMIC_DATA."$ctrl_EngDeng" )
      wire#w2
      S_Coil( #DYNAMIC_DATA.status_Energising )
   END_RUNG
   RUNG wire#powerrail
      Contact( #DYNAMIC_DATA.mode_Reset )
   END_RUNG wire#w1
   RUNG wire#w2
      R_Coil( #DYNAMIC_DATA.status_Deenergising )
   END_RUNG
   RUNG wire#w2
      Move(in := #STATIC_DATA.TIME_ENG_MAX, out1 => #DYNAMIC_DATA.actual_Operating_Timer)
   END_RUNG
   RUNG wire#w2
      { S7_Templates := "SrcType := Real" } LT_Contact(in1 := #STATIC_DATA.TIME_ENG_MAX, in2 := #k_TIME_OP_MIN)
      Move(in := #k_TIME_OP_MIN, out1 => #DYNAMIC_DATA.actual_Operating_Timer)
   END_RUNG
   // the same network as SCL:
   #_w1 := NOT #DYNAMIC_DATA.status_Fault AND #DYNAMIC_DATA."$ctrl_EngDeng" AND NOT #DYNAMIC_DATA."$pret_eng";   // rising edge of #DYNAMIC_DATA."$ctrl_EngDeng"
   #DYNAMIC_DATA."$pret_eng" := #DYNAMIC_DATA."$ctrl_EngDeng";
   #_w2 := (#_w1 OR #DYNAMIC_DATA.mode_Reset) AND #DYNAMIC_DATA."$ctrl_EngDeng";
   IF #_w2 THEN
       #DYNAMIC_DATA.status_Energising := TRUE;
       #DYNAMIC_DATA.status_Deenergising := FALSE;
       #DYNAMIC_DATA.actual_Operating_Timer := #STATIC_DATA.TIME_ENG_MAX;
   END_IF;
   IF #_w2 AND (#STATIC_DATA.TIME_ENG_MAX < #k_TIME_OP_MIN) THEN
       #DYNAMIC_DATA.actual_Operating_Timer := #k_TIME_OP_MIN;
   END_IF;
END_REGION

REGION Network 32: Check for change of state request — Deenergising
   // ▀▀▀▀▀▀▀▀▀▀▀▀▀▀▀▀▀▀▀▀▀▀▀▀▀▀▀▀▀▀▀▀▀▀▀▀▀▀▀▀▀▀▀▀
   // If a change of state is detected on ctrl_EngDeng, in this case a falling edge indicating the
   // valve has been requested to change from an energised to a deenergised state, the status of the
   // valve is set to deenergising and the deenergising operation time is loaded into the operation 
   // timer.
   // 
   // If the deenergising operation time is less than k_TIME_OP_MIN (210ms), the 
   // actual_Operating_Timer is set to k_TIME_OP_MIN. This ensure that at least one timing pulse is 
   // required, before the timer reaches a value of zero (i.e. at least one controller cycle will be 
   // required).
   // 
   // If the valve is in a fault condition (status_Fault = true), the change of state is not evaluated
   // until the fault condition has cleared
   // 
   // Note: the timer is also triggered if the Reset signal is received and the valve is requested to be 
   //            deenergised
   // ▄▄▄▄▄▄▄▄▄▄▄▄▄▄▄▄▄▄▄▄▄▄▄▄▄▄▄▄▄▄▄▄▄▄▄▄▄▄▄▄▄▄▄▄
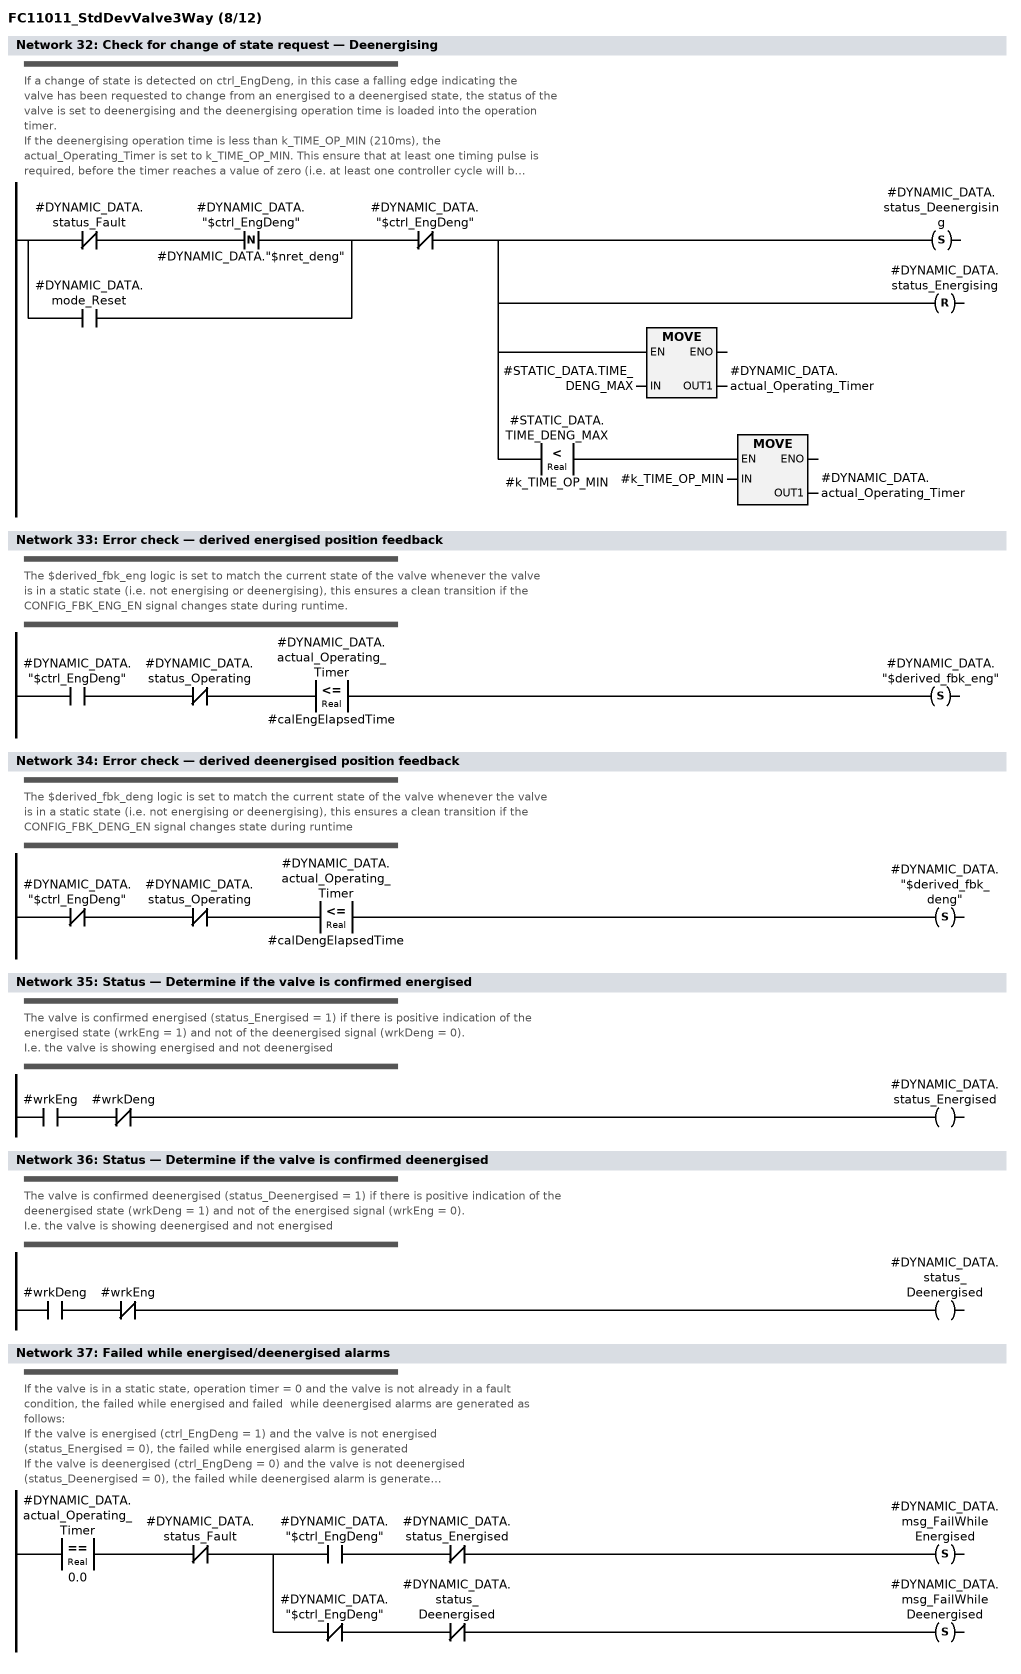
   RUNG wire#powerrail
      I_Contact( #DYNAMIC_DATA.status_Fault )
      N_Contact(operand := #DYNAMIC_DATA."$ctrl_EngDeng", bit := #DYNAMIC_DATA."$nret_deng")
      wire#w1
      I_Contact( #DYNAMIC_DATA."$ctrl_EngDeng" )
      wire#w2
      S_Coil( #DYNAMIC_DATA.status_Deenergising )
   END_RUNG
   RUNG wire#powerrail
      Contact( #DYNAMIC_DATA.mode_Reset )
   END_RUNG wire#w1
   RUNG wire#w2
      R_Coil( #DYNAMIC_DATA.status_Energising )
   END_RUNG
   RUNG wire#w2
      Move(in := #STATIC_DATA.TIME_DENG_MAX, out1 => #DYNAMIC_DATA.actual_Operating_Timer)
   END_RUNG
   RUNG wire#w2
      { S7_Templates := "SrcType := Real" } LT_Contact(in1 := #STATIC_DATA.TIME_DENG_MAX, in2 := #k_TIME_OP_MIN)
      Move(in := #k_TIME_OP_MIN, out1 => #DYNAMIC_DATA.actual_Operating_Timer)
   END_RUNG
   // the same network as SCL:
   #_w1 := NOT #DYNAMIC_DATA.status_Fault AND NOT #DYNAMIC_DATA."$ctrl_EngDeng" AND #DYNAMIC_DATA."$nret_deng";   // falling edge of #DYNAMIC_DATA."$ctrl_EngDeng"
   #DYNAMIC_DATA."$nret_deng" := #DYNAMIC_DATA."$ctrl_EngDeng";
   #_w2 := (#_w1 OR #DYNAMIC_DATA.mode_Reset) AND NOT #DYNAMIC_DATA."$ctrl_EngDeng";
   IF #_w2 THEN
       #DYNAMIC_DATA.status_Deenergising := TRUE;
       #DYNAMIC_DATA.status_Energising := FALSE;
       #DYNAMIC_DATA.actual_Operating_Timer := #STATIC_DATA.TIME_DENG_MAX;
   END_IF;
   IF #_w2 AND (#STATIC_DATA.TIME_DENG_MAX < #k_TIME_OP_MIN) THEN
       #DYNAMIC_DATA.actual_Operating_Timer := #k_TIME_OP_MIN;
   END_IF;
END_REGION

REGION Network 33: Error check — derived energised position feedback
   // ▀▀▀▀▀▀▀▀▀▀▀▀▀▀▀▀▀▀▀▀▀▀▀▀▀▀▀▀▀▀▀▀▀▀▀▀▀▀▀▀▀▀▀▀
   // The $derived_fbk_eng logic is set to match the current state of the valve whenever the valve
   // is in a static state (i.e. not energising or deenergising), this ensures a clean transition if the 
   // CONFIG_FBK_ENG_EN signal changes state during runtime.
   // ▄▄▄▄▄▄▄▄▄▄▄▄▄▄▄▄▄▄▄▄▄▄▄▄▄▄▄▄▄▄▄▄▄▄▄▄▄▄▄▄▄▄▄▄
   RUNG wire#powerrail
      Contact( #DYNAMIC_DATA."$ctrl_EngDeng" )
      I_Contact( #DYNAMIC_DATA.status_Operating )
      { S7_Templates := "SrcType := Real" } LE_Contact(in1 := #DYNAMIC_DATA.actual_Operating_Timer, in2 := #calEngElapsedTime)
      S_Coil( #DYNAMIC_DATA."$derived_fbk_eng" )
   END_RUNG
   // the same network as SCL:
   IF #DYNAMIC_DATA."$ctrl_EngDeng" AND NOT #DYNAMIC_DATA.status_Operating AND (#DYNAMIC_DATA.actual_Operating_Timer <= #calEngElapsedTime) THEN
       #DYNAMIC_DATA."$derived_fbk_eng" := TRUE;
   END_IF;
END_REGION

REGION Network 34: Error check — derived deenergised position feedback
   // ▀▀▀▀▀▀▀▀▀▀▀▀▀▀▀▀▀▀▀▀▀▀▀▀▀▀▀▀▀▀▀▀▀▀▀▀▀▀▀▀▀▀▀▀
   // The $derived_fbk_deng logic is set to match the current state of the valve whenever the valve
   // is in a static state (i.e. not energising or deenergising), this ensures a clean transition if the 
   // CONFIG_FBK_DENG_EN signal changes state during runtime
   // ▄▄▄▄▄▄▄▄▄▄▄▄▄▄▄▄▄▄▄▄▄▄▄▄▄▄▄▄▄▄▄▄▄▄▄▄▄▄▄▄▄▄▄▄
   RUNG wire#powerrail
      I_Contact( #DYNAMIC_DATA."$ctrl_EngDeng" )
      I_Contact( #DYNAMIC_DATA.status_Operating )
      { S7_Templates := "SrcType := Real" } LE_Contact(in1 := #DYNAMIC_DATA.actual_Operating_Timer, in2 := #calDengElapsedTime)
      S_Coil( #DYNAMIC_DATA."$derived_fbk_deng" )
   END_RUNG
   // the same network as SCL:
   IF NOT #DYNAMIC_DATA."$ctrl_EngDeng" AND NOT #DYNAMIC_DATA.status_Operating AND (#DYNAMIC_DATA.actual_Operating_Timer <= #calDengElapsedTime) THEN
       #DYNAMIC_DATA."$derived_fbk_deng" := TRUE;
   END_IF;
END_REGION

REGION Network 35: Status — Determine if the valve is confirmed energised
   // ▀▀▀▀▀▀▀▀▀▀▀▀▀▀▀▀▀▀▀▀▀▀▀▀▀▀▀▀▀▀▀▀▀▀▀▀▀▀▀▀▀▀▀▀
   // The valve is confirmed energised (status_Energised = 1) if there is positive indication of the 
   // energised state (wrkEng = 1) and not of the deenergised signal (wrkDeng = 0). 
   // 
   // I.e. the valve is showing energised and not deenergised
   // ▄▄▄▄▄▄▄▄▄▄▄▄▄▄▄▄▄▄▄▄▄▄▄▄▄▄▄▄▄▄▄▄▄▄▄▄▄▄▄▄▄▄▄▄
   RUNG wire#powerrail
      Contact( #wrkEng )
      I_Contact( #wrkDeng )
      Coil( #DYNAMIC_DATA.status_Energised )
   END_RUNG
   // the same network as SCL:
   #DYNAMIC_DATA.status_Energised := #wrkEng AND NOT #wrkDeng;
END_REGION

REGION Network 36: Status — Determine if the valve is confirmed deenergised
   // ▀▀▀▀▀▀▀▀▀▀▀▀▀▀▀▀▀▀▀▀▀▀▀▀▀▀▀▀▀▀▀▀▀▀▀▀▀▀▀▀▀▀▀▀
   // The valve is confirmed deenergised (status_Deenergised = 1) if there is positive indication of the 
   // deenergised state (wrkDeng = 1) and not of the energised signal (wrkEng = 0). 
   // 
   // I.e. the valve is showing deenergised and not energised
   // ▄▄▄▄▄▄▄▄▄▄▄▄▄▄▄▄▄▄▄▄▄▄▄▄▄▄▄▄▄▄▄▄▄▄▄▄▄▄▄▄▄▄▄▄
   RUNG wire#powerrail
      Contact( #wrkDeng )
      I_Contact( #wrkEng )
      Coil( #DYNAMIC_DATA.status_Deenergised )
   END_RUNG
   // the same network as SCL:
   #DYNAMIC_DATA.status_Deenergised := #wrkDeng AND NOT #wrkEng;
END_REGION

REGION Network 37: Failed while energised/deenergised alarms
   // ▀▀▀▀▀▀▀▀▀▀▀▀▀▀▀▀▀▀▀▀▀▀▀▀▀▀▀▀▀▀▀▀▀▀▀▀▀▀▀▀▀▀▀▀
   // If the valve is in a static state, operation timer = 0 and the valve is not already in a fault
   // condition, the failed while energised and failed  while deenergised alarms are generated as 
   // follows:
   // 
   // If the valve is energised (ctrl_EngDeng = 1) and the valve is not energised 
   // (status_Energised = 0), the failed while energised alarm is generated
   // 
   // If the valve is deenergised (ctrl_EngDeng = 0) and the valve is not deenergised 
   // (status_Deenergised = 0), the failed while deenergised alarm is generated
   // ▄▄▄▄▄▄▄▄▄▄▄▄▄▄▄▄▄▄▄▄▄▄▄▄▄▄▄▄▄▄▄▄▄▄▄▄▄▄▄▄▄▄▄▄
   RUNG wire#powerrail
      { S7_Templates := "SrcType := Real" } EQ_Contact(in1 := #DYNAMIC_DATA.actual_Operating_Timer, in2 := 0.0)
      I_Contact( #DYNAMIC_DATA.status_Fault )
      wire#w1
      Contact( #DYNAMIC_DATA."$ctrl_EngDeng" )
      I_Contact( #DYNAMIC_DATA.status_Energised )
      S_Coil( #DYNAMIC_DATA.msg_FailWhileEnergised )
   END_RUNG
   RUNG wire#w1
      I_Contact( #DYNAMIC_DATA."$ctrl_EngDeng" )
      I_Contact( #DYNAMIC_DATA.status_Deenergised )
      S_Coil( #DYNAMIC_DATA.msg_FailWhileDeenergised )
   END_RUNG
   // the same network as SCL:
   #_w1 := (#DYNAMIC_DATA.actual_Operating_Timer = 0.0) AND NOT #DYNAMIC_DATA.status_Fault;
   IF #_w1 AND #DYNAMIC_DATA."$ctrl_EngDeng" AND NOT #DYNAMIC_DATA.status_Energised THEN
       #DYNAMIC_DATA.msg_FailWhileEnergised := TRUE;
   END_IF;
   IF #_w1 AND NOT #DYNAMIC_DATA."$ctrl_EngDeng" AND NOT #DYNAMIC_DATA.status_Deenergised THEN
       #DYNAMIC_DATA.msg_FailWhileDeenergised := TRUE;
   END_IF;
END_REGION

REGION Network 38: Operation timer and Failed to energise/deenergise alarms
   // ▀▀▀▀▀▀▀▀▀▀▀▀▀▀▀▀▀▀▀▀▀▀▀▀▀▀▀▀▀▀▀▀▀▀▀▀▀▀▀▀▀▀▀▀
   // If the valve is energising or deenergising decrement the current operation timer value on each 
   // 200ms pulse.
   // 
   // If the timer reaches zero, and the valve is energising, generate the failed to energise alarm.
   // 
   // If the timer reaches zero, and the valve is deenergising, generate the failed to deenergise alarm
   // ▄▄▄▄▄▄▄▄▄▄▄▄▄▄▄▄▄▄▄▄▄▄▄▄▄▄▄▄▄▄▄▄▄▄▄▄▄▄▄▄▄▄▄▄
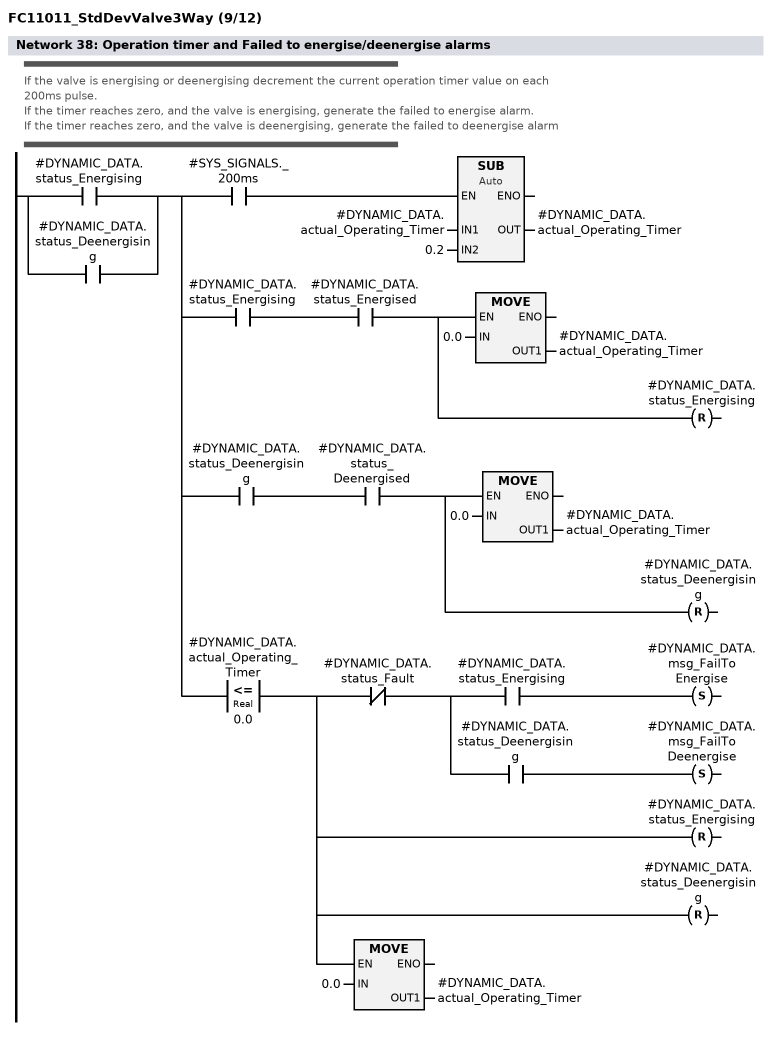
   RUNG wire#powerrail
      Contact( #DYNAMIC_DATA.status_Energising )
      wire#w1
      Contact( #SYS_SIGNALS._200ms )
      Sub(in1 := #DYNAMIC_DATA.actual_Operating_Timer, in2 := 0.2, out => #DYNAMIC_DATA.actual_Operating_Timer)
   END_RUNG
   RUNG wire#powerrail
      Contact( #DYNAMIC_DATA.status_Deenergising )
   END_RUNG wire#w1
   RUNG wire#w1
      Contact( #DYNAMIC_DATA.status_Energising )
      Contact( #DYNAMIC_DATA.status_Energised )
      wire#w2
      Move(in := 0.0, out1 => #DYNAMIC_DATA.actual_Operating_Timer)
   END_RUNG
   RUNG wire#w2
      R_Coil( #DYNAMIC_DATA.status_Energising )
   END_RUNG
   RUNG wire#w1
      Contact( #DYNAMIC_DATA.status_Deenergising )
      Contact( #DYNAMIC_DATA.status_Deenergised )
      wire#w3
      Move(in := 0.0, out1 => #DYNAMIC_DATA.actual_Operating_Timer)
   END_RUNG
   RUNG wire#w3
      R_Coil( #DYNAMIC_DATA.status_Deenergising )
   END_RUNG
   RUNG wire#w1
      { S7_Templates := "SrcType := Real" } LE_Contact(in1 := #DYNAMIC_DATA.actual_Operating_Timer, in2 := 0.0)
      wire#w4
      I_Contact( #DYNAMIC_DATA.status_Fault )
      wire#w5
      Contact( #DYNAMIC_DATA.status_Energising )
      S_Coil( #DYNAMIC_DATA.msg_FailToEnergise )
   END_RUNG
   RUNG wire#w5
      Contact( #DYNAMIC_DATA.status_Deenergising )
      S_Coil( #DYNAMIC_DATA.msg_FailToDeenergise )
   END_RUNG
   RUNG wire#w4
      R_Coil( #DYNAMIC_DATA.status_Energising )
   END_RUNG
   RUNG wire#w4
      R_Coil( #DYNAMIC_DATA.status_Deenergising )
   END_RUNG
   RUNG wire#w4
      Move(in := 0.0, out1 => #DYNAMIC_DATA.actual_Operating_Timer)
   END_RUNG
   // the same network as SCL:
   #_w1 := #DYNAMIC_DATA.status_Energising OR #DYNAMIC_DATA.status_Deenergising;
   IF #_w1 AND #SYS_SIGNALS._200ms THEN
       #DYNAMIC_DATA.actual_Operating_Timer := #DYNAMIC_DATA.actual_Operating_Timer - 0.2;
   END_IF;
   IF #_w1 AND #DYNAMIC_DATA.status_Energising AND #DYNAMIC_DATA.status_Energised THEN
       #DYNAMIC_DATA.actual_Operating_Timer := 0.0;
       #DYNAMIC_DATA.status_Energising := FALSE;
   END_IF;
   IF #_w1 AND #DYNAMIC_DATA.status_Deenergising AND #DYNAMIC_DATA.status_Deenergised THEN
       #DYNAMIC_DATA.actual_Operating_Timer := 0.0;
       #DYNAMIC_DATA.status_Deenergising := FALSE;
   END_IF;
   #_w2 := #_w1 AND (#DYNAMIC_DATA.actual_Operating_Timer <= 0.0);
   #_w3 := #_w2 AND NOT #DYNAMIC_DATA.status_Fault;
   IF #_w3 AND #DYNAMIC_DATA.status_Energising THEN #DYNAMIC_DATA.msg_FailToEnergise := TRUE; END_IF;
   IF #_w3 AND #DYNAMIC_DATA.status_Deenergising THEN #DYNAMIC_DATA.msg_FailToDeenergise := TRUE; END_IF;
   IF #_w2 THEN
       #DYNAMIC_DATA.status_Energising := FALSE;
       #DYNAMIC_DATA.status_Deenergising := FALSE;
       #DYNAMIC_DATA.actual_Operating_Timer := 0.0;
   END_IF;
END_REGION

REGION Network 39: Calculate last operation timer value
   // ▀▀▀▀▀▀▀▀▀▀▀▀▀▀▀▀▀▀▀▀▀▀▀▀▀▀▀▀▀▀▀▀▀▀▀▀▀▀▀▀▀▀▀▀
   // Stores that last good operation timer elapsed time, this is the elapsed value of the 
   // actual_Operating_Timer when the valve achieved the correct position. The result is subtracted
   // from the TIME_ENG/DENG_MAX value to give the true time to achieve position. The result
   // is stored in actual_Last_Op_Time
   // 
   // If the valve were energising, then actual_Last_Op_Time is calculated as follows:
   // 
   // ┌───────────────────────────────┐
   // │actual_Last_Op_Time = TIME_ENG_MAX ─ actual_Operating_Timer    │
   // └───────────────────────────────┘
   // 
   // If the valve were deenergising, then actual_Last_Op_Time is calculated as follows:
   // 
   // ┌────────────────────────────────┐
   // │actual_Last_Op_Time = TIME_DENG_MAX ─ actual_Operating_Timer     │
   // └────────────────────────────────┘
   // 
   // If the valve either fails to energise or fails to deenergise, then actual_Last_Op_Time is set 
   // to -1.0 to indicate a fault state.
   // ▄▄▄▄▄▄▄▄▄▄▄▄▄▄▄▄▄▄▄▄▄▄▄▄▄▄▄▄▄▄▄▄▄▄▄▄▄▄▄▄▄▄▄▄
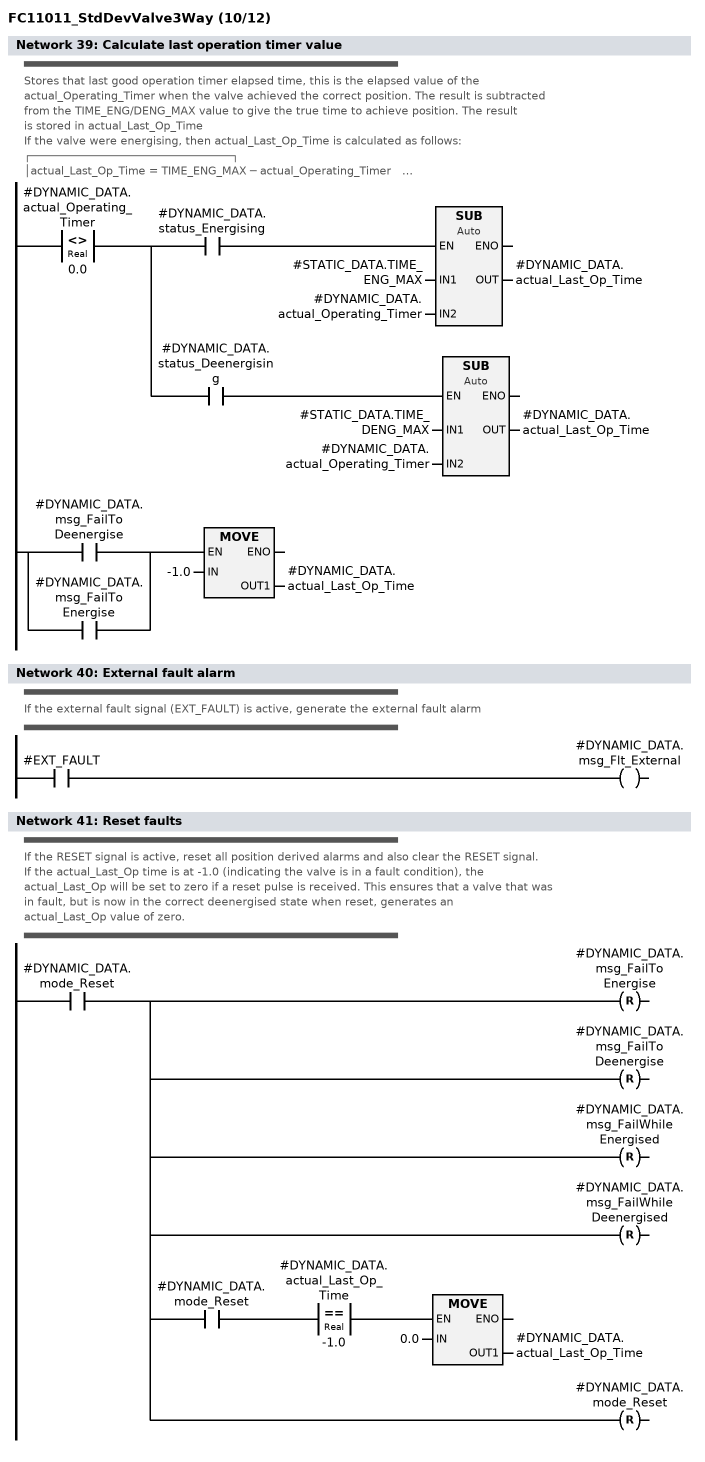
   RUNG wire#powerrail
      { S7_Templates := "SrcType := Real" } NE_Contact(in1 := #DYNAMIC_DATA.actual_Operating_Timer, in2 := 0.0)
      wire#w1
      Contact( #DYNAMIC_DATA.status_Energising )
      Sub(in1 := #STATIC_DATA.TIME_ENG_MAX, in2 := #DYNAMIC_DATA.actual_Operating_Timer, out => #DYNAMIC_DATA.actual_Last_Op_Time)
   END_RUNG
   RUNG wire#w1
      Contact( #DYNAMIC_DATA.status_Deenergising )
      Sub(in1 := #STATIC_DATA.TIME_DENG_MAX, in2 := #DYNAMIC_DATA.actual_Operating_Timer, out => #DYNAMIC_DATA.actual_Last_Op_Time)
   END_RUNG
   RUNG wire#powerrail
      Contact( #DYNAMIC_DATA.msg_FailToDeenergise )
      wire#w2
      Move(in := -1.0, out1 => #DYNAMIC_DATA.actual_Last_Op_Time)
   END_RUNG
   RUNG wire#powerrail
      Contact( #DYNAMIC_DATA.msg_FailToEnergise )
   END_RUNG wire#w2
   // the same network as SCL:
   #_w1 := #DYNAMIC_DATA.actual_Operating_Timer <> 0.0;
   IF #_w1 AND #DYNAMIC_DATA.status_Energising THEN
       #DYNAMIC_DATA.actual_Last_Op_Time := #STATIC_DATA.TIME_ENG_MAX - #DYNAMIC_DATA.actual_Operating_Timer;
   END_IF;
   IF #_w1 AND #DYNAMIC_DATA.status_Deenergising THEN
       #DYNAMIC_DATA.actual_Last_Op_Time := #STATIC_DATA.TIME_DENG_MAX - #DYNAMIC_DATA.actual_Operating_Timer;
   END_IF;
   IF #DYNAMIC_DATA.msg_FailToDeenergise OR #DYNAMIC_DATA.msg_FailToEnergise THEN
       #DYNAMIC_DATA.actual_Last_Op_Time := -1.0;
   END_IF;
END_REGION

REGION Network 40: External fault alarm
   // ▀▀▀▀▀▀▀▀▀▀▀▀▀▀▀▀▀▀▀▀▀▀▀▀▀▀▀▀▀▀▀▀▀▀▀▀▀▀▀▀▀▀▀▀
   // If the external fault signal (EXT_FAULT) is active, generate the external fault alarm
   // ▄▄▄▄▄▄▄▄▄▄▄▄▄▄▄▄▄▄▄▄▄▄▄▄▄▄▄▄▄▄▄▄▄▄▄▄▄▄▄▄▄▄▄▄
   RUNG wire#powerrail
      Contact( #EXT_FAULT )
      Coil( #DYNAMIC_DATA.msg_Flt_External )
   END_RUNG
   // the same network as SCL:
   #DYNAMIC_DATA.msg_Flt_External := #EXT_FAULT;
END_REGION

REGION Network 41: Reset faults
   // ▀▀▀▀▀▀▀▀▀▀▀▀▀▀▀▀▀▀▀▀▀▀▀▀▀▀▀▀▀▀▀▀▀▀▀▀▀▀▀▀▀▀▀▀
   // If the RESET signal is active, reset all position derived alarms and also clear the RESET signal.
   // 
   // If the actual_Last_Op time is at -1.0 (indicating the valve is in a fault condition), the 
   // actual_Last_Op will be set to zero if a reset pulse is received. This ensures that a valve that was 
   // in fault, but is now in the correct deenergised state when reset, generates an 
   // actual_Last_Op value of zero.
   // ▄▄▄▄▄▄▄▄▄▄▄▄▄▄▄▄▄▄▄▄▄▄▄▄▄▄▄▄▄▄▄▄▄▄▄▄▄▄▄▄▄▄▄▄
   RUNG wire#powerrail
      Contact( #DYNAMIC_DATA.mode_Reset )
      wire#w1
      R_Coil( #DYNAMIC_DATA.msg_FailToEnergise )
   END_RUNG
   RUNG wire#w1
      R_Coil( #DYNAMIC_DATA.msg_FailToDeenergise )
   END_RUNG
   RUNG wire#w1
      R_Coil( #DYNAMIC_DATA.msg_FailWhileEnergised )
   END_RUNG
   RUNG wire#w1
      R_Coil( #DYNAMIC_DATA.msg_FailWhileDeenergised )
   END_RUNG
   RUNG wire#w1
      Contact( #DYNAMIC_DATA.mode_Reset )
      { S7_Templates := "SrcType := Real" } EQ_Contact(in1 := #DYNAMIC_DATA.actual_Last_Op_Time, in2 := -1.0)
      Move(in := 0.0, out1 => #DYNAMIC_DATA.actual_Last_Op_Time)
   END_RUNG
   RUNG wire#w1
      R_Coil( #DYNAMIC_DATA.mode_Reset )
   END_RUNG
   // the same network as SCL:
   IF #DYNAMIC_DATA.mode_Reset THEN
       #DYNAMIC_DATA.msg_FailToEnergise := FALSE;
       #DYNAMIC_DATA.msg_FailToDeenergise := FALSE;
       #DYNAMIC_DATA.msg_FailWhileEnergised := FALSE;
       #DYNAMIC_DATA.msg_FailWhileDeenergised := FALSE;
   END_IF;
   IF #DYNAMIC_DATA.mode_Reset AND #DYNAMIC_DATA.mode_Reset AND (#DYNAMIC_DATA.actual_Last_Op_Time = (-1.0)) THEN
       #DYNAMIC_DATA.actual_Last_Op_Time := 0.0;
   END_IF;
   IF #DYNAMIC_DATA.mode_Reset THEN #DYNAMIC_DATA.mode_Reset := FALSE; END_IF;
END_REGION

